HMI tags "Planchadora1"
   "Planchadora1_EstadoSsDer" : Byte = PLC Planchadora1.EstadoSsDer, 1 s
   "Planchadora1_EstadoSsIzq" : Byte = PLC Planchadora1.EstadoSsIzq, 1 s
   "Planchadora1_EstadoSSMed" : Byte = PLC Planchadora1.EstadoSSMed, 1 s
   "Planchadora1_FactorCorrRend" : Real = PLC Planchadora1.FactorCorrRend, 1 s
   "Planchadora1_FechaHoraPLC" : DTL = PLC Planchadora1.FechaHoraPLC, 1 s
   "Planchadora1_Operadores{1}_Estado" : Bool = PLC Planchadora1.Operadores[1].Estado, 1 s
   "Planchadora1_Operadores{1}_Produccion" : DInt = PLC Planchadora1.Operadores[1].Produccion, 1 s
   "Planchadora1_Operadores{1}_Rendimiento" : DInt = PLC Planchadora1.Operadores[1].Rendimiento, 1 s
   "Planchadora1_Operadores{1}_RendPesado" : DInt = PLC Planchadora1.Operadores[1].RendPesado, 1 s
   "Planchadora1_Operadores{1}_Tiempo" : DInt = PLC Planchadora1.Operadores[1].Tiempo, 1 s
   "Planchadora1_Operadores{10}_Estado" : Bool = PLC Planchadora1.Operadores[10].Estado, 1 s
   "Planchadora1_Operadores{10}_Produccion" : DInt = PLC Planchadora1.Operadores[10].Produccion, 1 s
   "Planchadora1_Operadores{10}_Rendimiento" : DInt = PLC Planchadora1.Operadores[10].Rendimiento, 1 s
   "Planchadora1_Operadores{10}_RendPesado" : DInt = PLC Planchadora1.Operadores[10].RendPesado AT %DB1.DBD0, 1 s
   "Planchadora1_Operadores{10}_Tiempo" : DInt = PLC Planchadora1.Operadores[10].Tiempo, 1 s
   "Planchadora1_Operadores{2}_Estado" : Bool = PLC Planchadora1.Operadores[2].Estado, 1 s
   "Planchadora1_Operadores{2}_Produccion" : DInt = PLC Planchadora1.Operadores[2].Produccion, 1 s
   "Planchadora1_Operadores{2}_Rendimiento" : DInt = PLC Planchadora1.Operadores[2].Rendimiento, 1 s
   "Planchadora1_Operadores{2}_RendPesado" : DInt = PLC Planchadora1.Operadores[2].RendPesado AT %DB1.DBD0, 1 s
   "Planchadora1_Operadores{2}_Tiempo" : DInt = PLC Planchadora1.Operadores[2].Tiempo, 1 s
   "Planchadora1_Operadores{3}_Estado" : Bool = PLC Planchadora1.Operadores[3].Estado, 1 s
   "Planchadora1_Operadores{3}_Produccion" : DInt = PLC Planchadora1.Operadores[3].Produccion, 1 s
   "Planchadora1_Operadores{3}_Rendimiento" : DInt = PLC Planchadora1.Operadores[3].Rendimiento, 1 s
   "Planchadora1_Operadores{3}_RendPesado" : DInt = PLC Planchadora1.Operadores[3].RendPesado AT %DB1.DBD0, 1 s
   "Planchadora1_Operadores{3}_Tiempo" : DInt = PLC Planchadora1.Operadores[3].Tiempo, 1 s
   "Planchadora1_Operadores{4}_Estado" : Bool = PLC Planchadora1.Operadores[4].Estado, 1 s
   "Planchadora1_Operadores{4}_Produccion" : DInt = PLC Planchadora1.Operadores[4].Produccion, 1 s
   "Planchadora1_Operadores{4}_Rendimiento" : DInt = PLC Planchadora1.Operadores[4].Rendimiento, 1 s
   "Planchadora1_Operadores{4}_RendPesado" : DInt = PLC Planchadora1.Operadores[4].RendPesado AT %DB1.DBD0, 1 s
   "Planchadora1_Operadores{4}_Tiempo" : DInt = PLC Planchadora1.Operadores[4].Tiempo, 1 s
   "Planchadora1_Operadores{5}_Estado" : Bool = PLC Planchadora1.Operadores[4].Estado, 1 s
   "Planchadora1_Operadores{5}_Produccion" : DInt = PLC Planchadora1.Operadores[4].Produccion, 1 s
   "Planchadora1_Operadores{5}_Rendimiento" : DInt = PLC Planchadora1.Operadores[4].Rendimiento, 1 s
   "Planchadora1_Operadores{5}_RendPesado" : DInt = PLC Planchadora1.Operadores[4].RendPesado AT %DB1.DBD0, 1 s
   "Planchadora1_Operadores{5}_Tiempo" : DInt = PLC Planchadora1.Operadores[4].Tiempo, 1 s
   "Planchadora1_Operadores{6}_Estado" : Bool = PLC Planchadora1.Operadores[6].Estado, 1 s
   "Planchadora1_Operadores{6}_Produccion" : DInt = PLC Planchadora1.Operadores[6].Produccion, 1 s
   "Planchadora1_Operadores{6}_Rendimiento" : DInt = PLC Planchadora1.Operadores[6].Rendimiento, 1 s
   "Planchadora1_Operadores{6}_RendPesado" : DInt = PLC Planchadora1.Operadores[6].RendPesado AT %DB1.DBD0, 1 s
   "Planchadora1_Operadores{6}_Tiempo" : DInt = PLC Planchadora1.Operadores[6].Tiempo, 1 s
   "Planchadora1_Operadores{7}_Estado" : Bool = PLC Planchadora1.Operadores[6].Estado, 1 s
   "Planchadora1_Operadores{7}_Produccion" : DInt = PLC Planchadora1.Operadores[6].Produccion, 1 s
   "Planchadora1_Operadores{7}_Rendimiento" : DInt = PLC Planchadora1.Operadores[7].Rendimiento, 1 s
   "Planchadora1_Operadores{7}_RendPesado" : DInt = PLC Planchadora1.Operadores[6].RendPesado AT %DB1.DBD0, 1 s
   "Planchadora1_WeekDay" : USInt = PLC Planchadora1.FechaHoraPLC.WEEKDAY AT %DB1.DBX0.0, 1 s
   "Planchadora1_TiempoTotal" : DInt = PLC Planchadora1.TiempoTotal, 1 s
   "Planchadora1_Supervisores{4}_Tiempo" : DInt = PLC Planchadora1.Supervisores[4].Tiempo, 1 s
   "Planchadora1_Supervisores{4}_RendPesado" : DInt = PLC Planchadora1.Supervisores[4].RendPesado AT %DB1.DBD0, 1 s
   "Planchadora1_Supervisores{4}_Rendimiento" : DInt = PLC Planchadora1.Supervisores[4].Rendimiento, 1 s
   "Planchadora1_Supervisores{4}_Produccion" : DInt = PLC Planchadora1.Supervisores[4].Produccion, 1 s
   "Planchadora1_Supervisores{4}_Estado" : Bool = PLC Planchadora1.Supervisores[4].Estado, 1 s
   "Planchadora1_Supervisores{4}_Diadelasemana{7}_Salida" : Time_Of_Day = PLC Planchadora1.Supervisores[4].Diadelasemana[7].Salida, 1 h
   "Planchadora1_Supervisores{4}_Diadelasemana{7}_Entrada" : Time_Of_Day = PLC Planchadora1.Supervisores[4].Diadelasemana[7].Entrada, 1 h
   "Planchadora1_Supervisores{4}_Diadelasemana{7}_CantOp" : Int = PLC Planchadora1.Supervisores[4].Diadelasemana[7].CantOp, 1 s
   "Planchadora1_Supervisores{4}_Diadelasemana{6}_Salida" : Time_Of_Day = PLC Planchadora1.Supervisores[4].Diadelasemana[6].Salida, 1 h
   "Planchadora1_Supervisores{4}_Diadelasemana{6}_Entrada" : Time_Of_Day = PLC Planchadora1.Supervisores[4].Diadelasemana[6].Entrada, 1 h
   "Planchadora1_Supervisores{4}_Diadelasemana{3}_CantOp" : Int = PLC Planchadora1.Supervisores[4].Diadelasemana[3].CantOp, 1 s
   "Planchadora1_Supervisores{4}_Diadelasemana{3}_Entrada" : Time_Of_Day = PLC Planchadora1.Supervisores[4].Diadelasemana[3].Entrada, 1 h
   "Planchadora1_Supervisores{4}_Diadelasemana{3}_Salida" : Time_Of_Day = PLC Planchadora1.Supervisores[4].Diadelasemana[3].Salida, 1 h
   "Planchadora1_Supervisores{4}_Diadelasemana{4}_CantOp" : Int = PLC Planchadora1.Supervisores[4].Diadelasemana[4].CantOp, 1 s
   "Planchadora1_Supervisores{4}_Diadelasemana{4}_Entrada" : Time_Of_Day = PLC Planchadora1.Supervisores[4].Diadelasemana[4].Entrada, 1 h
   "Planchadora1_Supervisores{4}_Diadelasemana{4}_Salida" : Time_Of_Day = PLC Planchadora1.Supervisores[4].Diadelasemana[4].Salida, 1 h
   "Planchadora1_Supervisores{4}_Diadelasemana{5}_CantOp" : Int = PLC Planchadora1.Supervisores[4].Diadelasemana[5].CantOp, 1 s
   "Planchadora1_Supervisores{4}_Diadelasemana{5}_Entrada" : Time_Of_Day = PLC Planchadora1.Supervisores[4].Diadelasemana[5].Entrada, 1 h
   "Planchadora1_Supervisores{4}_Diadelasemana{5}_Salida" : Time_Of_Day = PLC Planchadora1.Supervisores[4].Diadelasemana[5].Salida, 1 h
   "Planchadora1_Supervisores{4}_Diadelasemana{6}_CantOp" : Int = PLC Planchadora1.Supervisores[4].Diadelasemana[6].CantOp, 1 s
   "Planchadora1_Supervisores{3}_Diadelasemana{6}_Salida" : Time_Of_Day = PLC Planchadora1.Supervisores[3].Diadelasemana[6].Salida, 1 h
   "Planchadora1_Supervisores{3}_Diadelasemana{7}_CantOp" : Int = PLC Planchadora1.Supervisores[3].Diadelasemana[7].CantOp, 1 s
   "Planchadora1_Supervisores{3}_Diadelasemana{7}_Entrda" : Time_Of_Day = PLC Planchadora1.Supervisores[3].Diadelasemana[7].Entrada, 1 h
   "Planchadora1_Supervisores{3}_Diadelasemana{7}_Salida" : Time_Of_Day = PLC Planchadora1.Supervisores[3].Diadelasemana[7].Salida, 1 h
   "Planchadora1_Supervisores{3}_Estado" : Bool = PLC Planchadora1.Supervisores[3].Estado, 1 s
   "Planchadora1_Supervisores{3}_Produccion" : DInt = PLC Planchadora1.Supervisores[3].Produccion, 1 s
   "Planchadora1_Supervisores{3}_Rendimiento" : DInt = PLC Planchadora1.Supervisores[3].Rendimiento, 1 s
   "Planchadora1_Supervisores{3}_RendPesado" : DInt = PLC Planchadora1.Supervisores[3].RendPesado AT %DB1.DBD0, 1 s
   "Planchadora1_Supervisores{3}_Tiempo" : DInt = PLC Planchadora1.Supervisores[3].Tiempo, 1 s
   "Planchadora1_Supervisores{4}_Diadelasemana{1}_CantOp" : Int = PLC Planchadora1.Supervisores[4].Diadelasemana[1].CantOp, 1 s
   "Planchadora1_Supervisores{4}_Diadelasemana{1}_Entrada" : Time_Of_Day = PLC Planchadora1.Supervisores[4].Diadelasemana[1].Entrada, 1 h
   "Planchadora1_Supervisores{4}_Diadelasemana{1}_Salida" : Time_Of_Day = PLC Planchadora1.Supervisores[4].Diadelasemana[1].Salida, 1 h
   "Planchadora1_Supervisores{4}_Diadelasemana{2}_CantOp" : Int = PLC Planchadora1.Supervisores[4].Diadelasemana[2].CantOp, 1 s
   "Planchadora1_Supervisores{4}_Diadelasemana{2}_Entrada" : Time_Of_Day = PLC Planchadora1.Supervisores[4].Diadelasemana[2].Entrada, 1 h
   "Planchadora1_Supervisores{4}_Diadelasemana{2}_Salida" : Time_Of_Day = PLC Planchadora1.Supervisores[4].Diadelasemana[2].Salida, 1 h
   "Planchadora1_Supervisores{3}_Diadelasemana{1}_Salida" : Time_Of_Day = PLC Planchadora1.Supervisores[3].Diadelasemana[1].Salida, 1 h
   "Planchadora1_Supervisores{3}_Diadelasemana{2}_CantOp" : Int = PLC Planchadora1.Supervisores[3].Diadelasemana[2].CantOp, 1 s
   "Planchadora1_Supervisores{3}_Diadelasemana{2}_Entrda" : Time_Of_Day = PLC Planchadora1.Supervisores[3].Diadelasemana[2].Entrada, 1 h
   "Planchadora1_Supervisores{3}_Diadelasemana{2}_Salida" : Time_Of_Day = PLC Planchadora1.Supervisores[3].Diadelasemana[2].Salida, 1 h
   "Planchadora1_Supervisores{3}_Diadelasemana{3}_CantOp" : Int = PLC Planchadora1.Supervisores[3].Diadelasemana[3].CantOp, 1 s
   "Planchadora1_Supervisores{3}_Diadelasemana{3}_Entrda" : Time_Of_Day = PLC Planchadora1.Supervisores[3].Diadelasemana[3].Entrada, 1 h
   "Planchadora1_Supervisores{3}_Diadelasemana{3}_Salida" : Time_Of_Day = PLC Planchadora1.Supervisores[3].Diadelasemana[3].Salida, 1 h
   "Planchadora1_Supervisores{3}_Diadelasemana{4}_CantOp" : Int = PLC Planchadora1.Supervisores[3].Diadelasemana[4].CantOp, 1 s
   "Planchadora1_Supervisores{3}_Diadelasemana{4}_Entrda" : Time_Of_Day = PLC Planchadora1.Supervisores[3].Diadelasemana[4].Entrada, 1 h
   "Planchadora1_Supervisores{3}_Diadelasemana{4}_Salida" : Time_Of_Day = PLC Planchadora1.Supervisores[3].Diadelasemana[4].Salida, 1 h
   "Planchadora1_Supervisores{3}_Diadelasemana{5}_CantOp" : Int = PLC Planchadora1.Supervisores[3].Diadelasemana[5].CantOp, 1 s
   "Planchadora1_Supervisores{3}_Diadelasemana{5}_Entrda" : Time_Of_Day = PLC Planchadora1.Supervisores[3].Diadelasemana[5].Entrada, 1 h
   "Planchadora1_Supervisores{3}_Diadelasemana{5}_Salida" : Time_Of_Day = PLC Planchadora1.Supervisores[3].Diadelasemana[5].Salida, 1 h
   "Planchadora1_Supervisores{3}_Diadelasemana{6}_CantOp" : Int = PLC Planchadora1.Supervisores[3].Diadelasemana[6].CantOp, 1 s
   "Planchadora1_Supervisores{3}_Diadelasemana{6}_Entrda" : Time_Of_Day = PLC Planchadora1.Supervisores[3].Diadelasemana[6].Entrada, 1 h
   "Planchadora1_Supervisores{2}_Diadelasemana{6}_Entrda" : Time_Of_Day = PLC Planchadora1.Supervisores[2].Diadelasemana[6].Entrada, 1 h
   "Planchadora1_Supervisores{2}_Diadelasemana{6}_Salida" : Time_Of_Day = PLC Planchadora1.Supervisores[2].Diadelasemana[6].Salida, 1 h
   "Planchadora1_Supervisores{2}_Diadelasemana{7}_CantOp" : Int = PLC Planchadora1.Supervisores[2].Diadelasemana[7].CantOp, 1 s
   "Planchadora1_Supervisores{2}_Diadelasemana{7}_Entrda" : Time_Of_Day = PLC Planchadora1.Supervisores[2].Diadelasemana[7].Entrada, 1 h
   "Planchadora1_Supervisores{2}_Diadelasemana{7}_Salida" : Time_Of_Day = PLC Planchadora1.Supervisores[2].Diadelasemana[7].Salida, 1 h
   "Planchadora1_Supervisores{2}_Estado" : Bool = PLC Planchadora1.Supervisores[2].Estado, 1 s
   "Planchadora1_Supervisores{2}_Produccion" : DInt = PLC Planchadora1.Supervisores[2].Produccion, 1 s
   "Planchadora1_Supervisores{2}_Rendimiento" : DInt = PLC Planchadora1.Supervisores[2].Rendimiento, 1 s
   "Planchadora1_Supervisores{2}_RendPesado" : DInt = PLC Planchadora1.Supervisores[2].RendPesado AT %DB1.DBD0, 1 s
   "Planchadora1_Supervisores{2}_Tiempo" : DInt = PLC Planchadora1.Supervisores[2].Tiempo, 1 s
   "Planchadora1_Supervisores{3}_Diadelasemana{1}_CantOp" : Int = PLC Planchadora1.Supervisores[3].Diadelasemana[1].CantOp, 1 s
   "Planchadora1_Supervisores{3}_Diadelasemana{1}_Entrda" : Time_Of_Day = PLC Planchadora1.Supervisores[3].Diadelasemana[1].Entrada, 1 h
   "Planchadora1_Supervisores{2}_Diadelasemana{2}_Entrda" : Time_Of_Day = PLC Planchadora1.Supervisores[2].Diadelasemana[2].Entrada, 1 h
   "Planchadora1_Supervisores{2}_Diadelasemana{2}_Salida" : Time_Of_Day = PLC Planchadora1.Supervisores[2].Diadelasemana[2].Salida, 1 h
   "Planchadora1_Supervisores{2}_Diadelasemana{3}_CantOp" : Int = PLC Planchadora1.Supervisores[2].Diadelasemana[3].CantOp, 1 s
   "Planchadora1_Supervisores{2}_Diadelasemana{3}_Entrda" : Time_Of_Day = PLC Planchadora1.Supervisores[2].Diadelasemana[3].Entrada, 1 h
   "Planchadora1_Supervisores{2}_Diadelasemana{3}_Salida" : Time_Of_Day = PLC Planchadora1.Supervisores[2].Diadelasemana[3].Salida, 1 h
   "Planchadora1_Supervisores{2}_Diadelasemana{4}_CantOp" : Int = PLC Planchadora1.Supervisores[2].Diadelasemana[4].CantOp, 1 s
   "Planchadora1_Supervisores{2}_Diadelasemana{4}_Entrda" : Time_Of_Day = PLC Planchadora1.Supervisores[2].Diadelasemana[4].Entrada, 1 h
   "Planchadora1_Supervisores{2}_Diadelasemana{4}_Salida" : Time_Of_Day = PLC Planchadora1.Supervisores[2].Diadelasemana[4].Salida, 1 h
   "Planchadora1_Supervisores{2}_Diadelasemana{5}_CantOp" : Int = PLC Planchadora1.Supervisores[2].Diadelasemana[5].CantOp, 1 s
   "Planchadora1_Supervisores{2}_Diadelasemana{5}_Entrda" : Time_Of_Day = PLC Planchadora1.Supervisores[2].Diadelasemana[5].Entrada, 1 h
   "Planchadora1_Supervisores{2}_Diadelasemana{5}_Salida" : Time_Of_Day = PLC Planchadora1.Supervisores[2].Diadelasemana[5].Salida, 1 h
   "Planchadora1_Supervisores{2}_Diadelasemana{6}_CantOp" : Int = PLC Planchadora1.Supervisores[2].Diadelasemana[6].CantOp, 1 s
   "Planchadora1_Supervisores{1}_Diadelasemana{6}_CantOp" : Int = PLC Planchadora1.Supervisores[1].Diadelasemana[6].CantOp, 1 s
   "Planchadora1_Supervisores{1}_Diadelasemana{6}_Entrda" : Time_Of_Day = PLC Planchadora1.Supervisores[1].Diadelasemana[6].Entrada, 1 h
   "Planchadora1_Supervisores{1}_Diadelasemana{6}_Salida" : Time_Of_Day = PLC Planchadora1.Supervisores[1].Diadelasemana[6].Salida, 1 h
   "Planchadora1_Supervisores{1}_Diadelasemana{7}_CantOp" : Int = PLC Planchadora1.Supervisores[1].Diadelasemana[7].CantOp, 1 s
   "Planchadora1_Supervisores{1}_Diadelasemana{7}_Entrda" : Time_Of_Day = PLC Planchadora1.Supervisores[1].Diadelasemana[7].Entrada, 1 h
   "Planchadora1_Supervisores{1}_Diadelasemana{7}_Salida" : Time_Of_Day = PLC Planchadora1.Supervisores[1].Diadelasemana[7].Salida, 1 h
   "Planchadora1_Supervisores{1}_Estado" : Bool = PLC Planchadora1.Supervisores[1].Estado, 1 s
   "Planchadora1_Supervisores{1}_Produccion" : DInt = PLC Planchadora1.Supervisores[1].Produccion, 1 s
   "Planchadora1_Supervisores{1}_Rendimiento" : DInt = PLC Planchadora1.Supervisores[1].Rendimiento, 1 s
   "Planchadora1_Supervisores{1}_RendPesado" : DInt = PLC Planchadora1.Supervisores[1].RendPesado AT %DB1.DBD0, 1 s
   "Planchadora1_Supervisores{1}_Tiempo" : DInt = PLC Planchadora1.Supervisores[1].Tiempo, 1 s
   "Planchadora1_Supervisores{2}_Diadelasemana{1}_CantOp" : Int = PLC Planchadora1.Supervisores[2].Diadelasemana[1].CantOp, 1 s
   "Planchadora1_Supervisores{2}_Diadelasemana{1}_Entrda" : Time_Of_Day = PLC Planchadora1.Supervisores[2].Diadelasemana[1].Entrada, 1 h
   "Planchadora1_Supervisores{2}_Diadelasemana{1}_Salida" : Time_Of_Day = PLC Planchadora1.Supervisores[2].Diadelasemana[1].Salida, 1 h
   "Planchadora1_Supervisores{2}_Diadelasemana{2}_CantOp" : Int = PLC Planchadora1.Supervisores[2].Diadelasemana[2].CantOp, 1 s
   "Planchadora1_Supervisores{1}_Diadelasemana{1}_CantOp" : Int = PLC Planchadora1.Supervisores[1].Diadelasemana[1].CantOp, 1 s
   "Planchadora1_Supervisores{1}_Diadelasemana{1}_Entrda" : Time_Of_Day = PLC Planchadora1.Supervisores[1].Diadelasemana[1].Entrada, 1 h
   "Planchadora1_Supervisores{1}_Diadelasemana{1}_Salida" : Time_Of_Day = PLC Planchadora1.Supervisores[1].Diadelasemana[1].Salida, 1 h
   "Planchadora1_Supervisores{1}_Diadelasemana{2}_CantOp" : Int = PLC Planchadora1.Supervisores[1].Diadelasemana[2].CantOp, 1 s
   "Planchadora1_Supervisores{1}_Diadelasemana{2}_Entrda" : Time_Of_Day = PLC Planchadora1.Supervisores[1].Diadelasemana[2].Entrada, 1 h
   "Planchadora1_Supervisores{1}_Diadelasemana{2}_Salida" : Time_Of_Day = PLC Planchadora1.Supervisores[1].Diadelasemana[2].Salida, 1 h
   "Planchadora1_Supervisores{1}_Diadelasemana{3}_CantOp" : Int = PLC Planchadora1.Supervisores[1].Diadelasemana[3].CantOp, 1 s
   "Planchadora1_Supervisores{1}_Diadelasemana{3}_Entrda" : Time_Of_Day = PLC Planchadora1.Supervisores[1].Diadelasemana[3].Entrada, 1 h
   "Planchadora1_Supervisores{1}_Diadelasemana{3}_Salida" : Time_Of_Day = PLC Planchadora1.Supervisores[1].Diadelasemana[3].Salida, 1 h
   "Planchadora1_Supervisores{1}_Diadelasemana{4}_CantOp" : Int = PLC Planchadora1.Supervisores[1].Diadelasemana[4].CantOp, 1 s
   "Planchadora1_Supervisores{1}_Diadelasemana{4}_Entrda" : Time_Of_Day = PLC Planchadora1.Supervisores[1].Diadelasemana[4].Entrada, 1 h
   "Planchadora1_Supervisores{1}_Diadelasemana{4}_Salida" : Time_Of_Day = PLC Planchadora1.Supervisores[1].Diadelasemana[4].Salida, 1 h
   "Planchadora1_Supervisores{1}_Diadelasemana{5}_CantOp" : Int = PLC Planchadora1.Supervisores[1].Diadelasemana[5].CantOp, 1 s
   "Planchadora1_Supervisores{1}_Diadelasemana{5}_Entrda" : Time_Of_Day = PLC Planchadora1.Supervisores[1].Diadelasemana[5].Entrada, 1 h
   "Planchadora1_Supervisores{1}_Diadelasemana{5}_Salida" : Time_Of_Day = PLC Planchadora1.Supervisores[1].Diadelasemana[5].Salida, 1 h
   "Planchadora1_Rendimiento_100" : Real = PLC Planchadora1.Rendimiento_100, 1 s
   "Planchadora1_Rendimiento_Amarillo" : Real = PLC Planchadora1.Productividad_Amarillo, 1 s
   "Planchadora1_Rendimiento_Rojo" : Real = PLC Planchadora1.Rendimiento_Rojo, 1 s
   "Planchadora1_Rendimiento_Verde" : Real = PLC Planchadora1.Productividad_Verde, 1 s
   "Planchadora1_RendimientoCada15" : DInt = PLC Planchadora1.RendimientoCada15, 1 s
   "Planchadora1_RendimientoTotal" : DInt = PLC Planchadora1.RendimientoTotal, 1 s
   "Planchadora1_RendPesado" : DInt = PLC Planchadora1.RendPesado AT %DB1.DBD0, 1 s
   "Planchadora1_RendPesado_100" : Real = PLC Planchadora1.RendPesado_100, 1 s
   "Planchadora1_SumaOperario" : Int = PLC Planchadora1.SumaOperario AT %DB1.DBX0.0, 10 s
      on ChangeValue: "S407_Act_IndicePLC"()
   "Planchadora1_Operadores{8}_Estado" : Bool = PLC Planchadora1.Operadores[8].Estado, 1 s
   "Planchadora1_Operadores{8}_Produccion" : DInt = PLC Planchadora1.Operadores[8].Produccion, 1 s
   "Planchadora1_Operadores{8}_Rendimiento" : DInt = PLC Planchadora1.Operadores[8].Rendimiento, 1 s
   "Planchadora1_Operadores{8}_RendPesado" : DInt = PLC Planchadora1.Operadores[8].RendPesado AT %DB1.DBD0, 1 s
   "Planchadora1_Operadores{8}_Tiempo" : DInt = PLC Planchadora1.Operadores[8].Tiempo, 1 s
   "Planchadora1_Operadores{9}_Estado" : Bool = PLC Planchadora1.Operadores[9].Estado, 1 s
   "Planchadora1_Operadores{9}_Produccion" : DInt = PLC Planchadora1.Operadores[9].Produccion, 1 s
   "Planchadora1_Operadores{9}_Rendimiento" : DInt = PLC Planchadora1.Operadores[9].Rendimiento, 1 s
   "Planchadora1_Operadores{9}_RendPesado" : DInt = PLC Planchadora1.Operadores[9].RendPesado AT %DB1.DBD0, 1 s
   "Planchadora1_Operadores{9}_Tiempo" : DInt = PLC Planchadora1.Operadores[9].Tiempo, 1 s
   "Planchadora1_Productividad" : DInt = PLC Planchadora1.Productividad, 1 s
   "Planchadora1_Productividad_100" : Real = PLC Planchadora1.Productividad_100, 1 s
   "Planchadora1_Productividad_Amarillo" : Real = PLC Planchadora1.Productividad_Amarillo, 1 s
   "Planchadora1_Productividad_Rojo" : Real = PLC Planchadora1.Productividad_Rojo, 1 s
   "Planchadora1_Productividad_Verde" : Real = PLC Planchadora1.Productividad_Verde, 1 s
   "Planchadora1_ProductividadCada15" : DInt = PLC Planchadora1.ProductividadCada15, 1 s
   "Planchadora1_ProductividadTotal" : DInt = PLC Planchadora1.ProductividadTotal, 1 s
   "Planchadora1_Rendimiento" : DInt = PLC Planchadora1.Rendimiento, 1 s
   "Planchadora1_Operadores{7}_Tiempo" : DInt = PLC Planchadora1.Operadores[7].Tiempo, 1 s

HMI tags "Planchadora2"
   "Planchadora2_WeekDay_Int" : Int AT %DB1.DBX0.0
   "Planchadora2_Supervisores{1}_Tiempo" : DInt = PLC Planchadora2.Supervisores[1].Tiempo, 1 s
   "Planchadora2_Supervisores{2}_Estado" : Bool = PLC Planchadora2.Supervisores[2].Estado, 1 s
   "Planchadora2_Supervisores{2}_Produccion" : DInt = PLC Planchadora2.Supervisores[2].Produccion, 1 s
   "Planchadora2_Supervisores{2}_Rendimiento" : DInt = PLC Planchadora2.Supervisores[2].Rendimiento, 1 s
   "Planchadora2_Supervisores{2}_RendPesado" : DInt = PLC Planchadora2.Supervisores[2].RendPesado AT %DB1.DBD0, 1 s
   "Planchadora2_Supervisores{2}_Tiempo" : DInt = PLC Planchadora2.Supervisores[2].Tiempo, 1 s
   "Planchadora2_Supervisores{3}_Estado" : Bool = PLC Planchadora2.Supervisores[3].Estado, 1 s
   "Planchadora2_Supervisores{3}_Produccion" : DInt = PLC Planchadora2.Supervisores[3].Produccion, 1 s
   "Planchadora2_Supervisores{3}_Rendimiento" : DInt = PLC Planchadora2.Supervisores[3].Rendimiento, 1 s
   "Planchadora2_Supervisores{3}_RendPesado" : DInt = PLC Planchadora2.Supervisores[3].RendPesado AT %DB1.DBD0, 1 s
   "Planchadora2_Supervisores{3}_Tiempo" : DInt = PLC Planchadora2.Supervisores[3].Tiempo, 1 s
   "Planchadora2_Supervisores{4}_Estado" : Bool = PLC Planchadora2.Supervisores[4].Estado, 1 s
   "Planchadora2_Supervisores{4}_Produccion" : DInt = PLC Planchadora2.Supervisores[4].Produccion, 1 s
   "Planchadora2_Supervisores{4}_Rendimiento" : DInt = PLC Planchadora2.Supervisores[4].Rendimiento, 1 s
   "Planchadora2_Supervisores{4}_RendPesado" : DInt = PLC Planchadora2.Supervisores[4].RendPesado AT %DB1.DBD0, 1 s
   "Planchadora2_Supervisores{4}_Tiempo" : DInt = PLC Planchadora2.Supervisores[4].Tiempo, 1 s
   "Planchadora2_TiempoTotal" : DInt = PLC Planchadora2.TiempoTotal, 1 s
   "Planchadora2_WeekDay" : USInt = PLC Planchadora2.FechaHoraPLC.WEEKDAY AT %DB1.DBB0, 1 s
   "Planchadora2_Operadores{9}_RendPesado" : DInt = PLC Planchadora2.Operadores[9].RendPesado AT %DB1.DBD0, 1 s
   "Planchadora2_Operadores{9}_Tiempo" : DInt = PLC Planchadora2.Operadores[9].Tiempo, 1 s
   "Planchadora2_Productividad_100" : Real = PLC Planchadora2.Productividad_100, 1 s
   "Planchadora2_ProductividadCada15" : DInt = PLC Planchadora2.ProductividadCada15, 1 s
   "Planchadora2_ProductividadTotal" : DInt = PLC Planchadora2.ProductividadTotal, 1 s
   "Planchadora2_Rendimiento_100" : Real = PLC Planchadora2.Rendimiento_100, 1 s
   "Planchadora2_RendimientoCada15" : DInt = PLC Planchadora2.RendimientoCada15, 1 s
   "Planchadora2_RendimientoTotal" : DInt = PLC Planchadora2.RendimientoTotal, 1 s
   "Planchadora2_RendPesado" : DInt = PLC Planchadora2.RendPesado AT %DB1.DBD0, 1 s
   "Planchadora2_RendPesado_100" : Real = PLC Planchadora2.RendPesado_100, 1 s
   "Planchadora2_SumaOperario" : Int = PLC Planchadora2.SumaOperario AT %DB1.DBX0.0, 1 s
   "Planchadora2_Supervisores{1}_Estado" : Bool = PLC Planchadora2.Supervisores[1].Estado, 1 s
   "Planchadora2_Supervisores{1}_Produccion" : DInt = PLC Planchadora2.Supervisores[1].Produccion, 1 s
   "Planchadora2_Supervisores{1}_Rendimiento" : DInt = PLC Planchadora2.Supervisores[1].Rendimiento, 1 s
   "Planchadora2_Supervisores{1}_RendPesado" : DInt = PLC Planchadora2.Supervisores[1].RendPesado AT %DB1.DBD0, 1 s
   "Planchadora2_Operadores{6}_Produccion" : DInt = PLC Planchadora2.Operadores[6].Produccion, 1 s
   "Planchadora2_Operadores{6}_Rendimiento" : DInt = PLC Planchadora2.Operadores[6].Rendimiento, 1 s
   "Planchadora2_Operadores{6}_RendPesado" : DInt = PLC Planchadora2.Operadores[6].RendPesado AT %DB1.DBD0, 1 s
   "Planchadora2_Operadores{6}_Tiempo" : DInt = PLC Planchadora2.Operadores[6].Tiempo, 1 s
   "Planchadora2_Operadores{7}_Estado" : Bool = PLC Planchadora2.Operadores[7].Estado, 1 s
   "Planchadora2_Operadores{7}_Produccion" : DInt = PLC Planchadora2.Operadores[7].Produccion, 1 s
   "Planchadora2_Operadores{7}_Rendimiento" : DInt = PLC Planchadora2.Operadores[7].Rendimiento, 1 s
   "Planchadora2_Operadores{7}_RendPesado" : DInt = PLC Planchadora2.Operadores[7].RendPesado AT %DB1.DBD0, 1 s
   "Planchadora2_Operadores{7}_Tiempo" : DInt = PLC Planchadora2.Operadores[7].Tiempo, 1 s
   "Planchadora2_Operadores{8}_Estado" : Bool = PLC Planchadora2.Operadores[8].Estado, 1 s
   "Planchadora2_Operadores{8}_Produccion" : DInt = PLC Planchadora2.Operadores[8].Produccion, 1 s
   "Planchadora2_Operadores{8}_Rendimiento" : DInt = PLC Planchadora2.Operadores[8].Rendimiento, 1 s
   "Planchadora2_Operadores{8}_RendPesado" : DInt = PLC Planchadora2.Operadores[8].RendPesado, 1 s
   "Planchadora2_Operadores{8}_Tiempo" : DInt = PLC Planchadora2.Operadores[8].Tiempo, 1 s
   "Planchadora2_Operadores{9}_Estado" : Bool = PLC Planchadora2.Operadores[9].Estado, 1 s
   "Planchadora2_Operadores{9}_Produccion" : DInt = PLC Planchadora2.Operadores[9].Produccion, 1 s
   "Planchadora2_Operadores{9}_Rendimiento" : DInt = PLC Planchadora2.Operadores[9].Rendimiento, 1 s
   "Planchadora2_Operadores{2}_RendPesado" : DInt = PLC Planchadora2.Operadores[2].RendPesado AT %DB1.DBD0, 1 s
   "Planchadora2_Operadores{2}_Tiempo" : DInt = PLC Planchadora2.Operadores[3].Tiempo, 1 s
   "Planchadora2_Operadores{3}_Estado" : Bool = PLC Planchadora2.Operadores[3].Estado, 1 s
   "Planchadora2_Operadores{3}_Produccion" : DInt = PLC Planchadora2.Operadores[3].Produccion, 1 s
   "Planchadora2_Operadores{3}_Rendimiento" : DInt = PLC Planchadora2.Operadores[3].Rendimiento, 1 s
   "Planchadora2_Operadores{3}_RendPesado" : DInt = PLC Planchadora2.Operadores[3].RendPesado AT %DB1.DBD0, 1 s
   "Planchadora2_Operadores{3}_Tiempo" : DInt = PLC Planchadora2.Operadores[3].Tiempo, 1 s
   "Planchadora2_Operadores{4}_Estado" : Bool = PLC Planchadora2.Operadores[4].Estado, 1 s
   "Planchadora2_Operadores{4}_Produccion" : DInt = PLC Planchadora2.Operadores[4].Produccion, 1 s
   "Planchadora2_Operadores{4}_Rendimiento" : DInt = PLC Planchadora2.Operadores[5].Rendimiento, 1 s
   "Planchadora2_Operadores{4}_RendPesado" : DInt = PLC Planchadora2.Operadores[5].RendPesado AT %DB1.DBD0, 1 s
   "Planchadora2_Operadores{4}_Tiempo" : DInt = PLC Planchadora2.Operadores[5].Tiempo, 1 s
   "Planchadora2_Operadores{5}_Estado" : Bool = PLC Planchadora2.Operadores[5].Estado, 1 s
   "Planchadora2_Operadores{5}_Produccion" : DInt = PLC Planchadora2.Operadores[5].Produccion, 1 s
   "Planchadora2_Operadores{5}_Rendimiento" : DInt = PLC Planchadora2.Operadores[5].Rendimiento, 1 s
   "Planchadora2_Operadores{5}_RendPesado" : DInt = PLC Planchadora2.Operadores[5].RendPesado AT %DB1.DBD0, 1 s
   "Planchadora2_Operadores{5}_Tiempo" : DInt = PLC Planchadora2.Operadores[5].Tiempo, 1 s
   "Planchadora2_Operadores{6}_Estado" : Bool = PLC Planchadora2.Operadores[6].Estado, 1 s
   "Planchadora2_EstadoSsIzq" : Byte = PLC Planchadora2.EstadoSsIzq, 1 s
   "Planchadora2_EstadoSSMed" : Byte = PLC Planchadora2.EstadoSSMed, 1 s
   "Planchadora2_Operadores{1}_Estado" : Bool = PLC Planchadora2.Operadores[1].Estado, 1 s
   "Planchadora2_Operadores{1}_Produccion" : DInt = PLC Planchadora2.Operadores[1].Produccion, 1 s
   "Planchadora2_Operadores{1}_Productividad" : DInt = PLC Planchadora2.Operadores[1].Productividad, 1 s
   "Planchadora2_Operadores{1}_Rendimiento" : DInt = PLC Planchadora2.Operadores[1].Rendimiento, 1 s
   "Planchadora2_Operadores{1}_RendPesado" : DInt = PLC Planchadora2.Operadores[1].RendPesado AT %DB1.DBD0, 1 s
   "Planchadora2_Operadores{1}_Tiempo" : DInt = PLC Planchadora2.Operadores[1].Tiempo, 1 s
   "Planchadora2_Operadores{10}_Estado" : Bool = PLC Planchadora2.Operadores[10].Estado, 1 s
   "Planchadora2_Operadores{10}_Produccion" : DInt = PLC Planchadora2.Operadores[10].Produccion, 1 s
   "Planchadora2_Operadores{10}_Rendimiento" : DInt = PLC Planchadora2.Operadores[10].Rendimiento, 1 s
   "Planchadora2_Operadores{10}_RendPesado" : DInt = PLC Planchadora2.Operadores[10].RendPesado AT %DB1.DBD0, 1 s
   "Planchadora2_Operadores{10}_Tiempo" : DInt = PLC Planchadora2.Operadores[10].Tiempo, 1 s
   "Planchadora2_Operadores{2}_Estado" : Bool = PLC Planchadora2.Operadores[2].Estado, 1 s
   "Planchadora2_Operadores{2}_Produccion" : DInt = PLC Planchadora2.Operadores[2].Produccion, 1 s
   "Planchadora2_Operadores{2}_Rendimiento" : DInt = PLC Planchadora2.Operadores[2].Rendimiento, 1 s
   "Plan2EnProd" : Bool = PLC Plan2EnProd AT %M4.3, 1 s
   "Planchadora2_EstadoSsDer" : Byte = PLC Planchadora2.EstadoSsDer, 1 s

HMI tags "Lavadora1"
   "Lav1_Programa" : Int AT 4x403158, 2 s
   "Lav1_Operador" : Int AT 4x403155, 2 s
      on ChangeValue: "S304_ActualizarOpEnPrincipal"(1)
   "Lav1_Alarma" : Bit AT 0x2057, 2 s
   "Lav1_CantRopa" : Int AT 4x403157, 2 s
   "Lav1_GrabarBDD" : Bit AT 0x3244, 1 s
      on ChangeValue: "S14_Write_data_Lav1"()
   "Lav1_FchFin_Ano" : Int AT 4x403172, 500 ms
   "Lav1_FchFin_Mes" : Int AT 4x403171, 500 ms
   "Lav1_FchFin_Dia" : Int AT 4x403170, 500 ms
   "Lav1_FchFin_Hr" : Int AT 4x403169, 500 ms
   "Lav1_FchFin_Min" : Int AT 4x403168, 500 ms
   "Lav1_FchFin_Seg" : Int AT 4x403167, 500 ms
   "Lav1_FchIni_Ano" : Int AT 4x403166, 1 s
   "Lav1_FchIni_Mes" : Int AT 4x403165, 1 s
   "Lav1_FchIni_Dia" : Int AT 4x403164, 1 s
   "Lav1_FchIni_Hr" : Int AT 4x403163, 1 s
   "Lav1_FchIni_Min" : Int AT 4x403162, 1 s
   "Lav1_FchIni_Seg" : Int AT 4x403161, 1 s
   "Lav1_Cliente_0" : Int AT 4x403160, 2 s
      on ChangeValue: "S104_ActualizarCliEmPrincipal"(1, 0)
   "Lav1_CicloValido" : Bit AT 0x3208, 100 ms
   "Lav1_Operador_Str" : WString[64], internal
   "Lav1_Cliente_1" : Int AT 4x403174, 2 s
      on ChangeValue: "S104_ActualizarCliEmPrincipal"(1, 1)
   "Lav1_Cliente_2" : Int AT 4x403176, 2 s
      on ChangeValue: "S104_ActualizarCliEmPrincipal"(1, 2)
   "Lav1_Fch_segs" : Int AT 4x404087, 500 ms
   "Lav1_Fch_Mins" : Int AT 4x404088, 500 ms
   "Lav1_Fch_Hr" : Int AT 4x404089, 500 ms
   "Lav1_Fch_Dia" : Int AT 4x404091, 500 ms
   "Lav1_Fch_Mes" : Int AT 4x404092, 500 ms
   "Lav1_Fch_Ano" : Int AT 4x404093, 500 ms
   "Lav1_Cliente_0_PLC" : Int AT 4x403159, 2 s
   "Lav1_Cliente_1_PLC" : Int AT 4x403173, 2 s
   "Lav1_Cliente_2_PLC" : Int AT 4x403175, 2 s
   "Lav1_Operador_PLC" : Int AT 4x403154, 2 s
      on ChangeValue: "S304_ActualizarOpEnPrincipal"(1)
   "Lav1_CantR_PLC" : Int AT 4x403156, 2 s
   "Lav1_AlarmaVibracion" : Bit AT 0x3390, 2 s
      on ChangeValue: "SA1_email_Vibr"(); "S40_Write_Fall1BDD"()
   "Lav1_EnCiclo" : Bit AT 0x3081, 1 s
      on ChangeValue: "SA3_Act_HoraFinEstPrincLav1"()
   "Lav1_CicloFinalizado" : Bit AT 0x3251, 2 s
   "Lav1_Ciclograbado" : Bit AT 0x3231, 1 s
   "Lav1_ComienzoCiclo" : Bit AT 0x3230, 1 s
   "Lav1_Falla" : Int AT 4x403183, 500 ms
   "Lav1_ConfFalla" : Bit AT 0x3252, 1 s
   "Lav1_PulsParadaPres" : Bit AT 0x3253, 1 s
      on ChangeValue: "S40_Write_Fall1BDD"()
   "Lav1_Cli_0_Str" : WString[64], internal
   "Lav1_Cli_1_Str" : WString[64], internal
   "Lav1_Cli_2_Str" : WString[64], internal
   "Lav1_FinEstimado_Panel" : DateTime, internal
   "Lav1_ProgAGrabar" : Int AT 4x401025, 2 s
   "Lav1_PulsParadaPres_1" : Bit AT 0x3254, 1 s
   "Lav1_Cont_IntentosGrabado" : Int, internal
   "Lav1_X0_iPres_SinAire" : Bit AT 0x2049, 1 s
   "Lav1_X1_iPres_Freno" : Bit AT 0x2050, 1 s
   "Lav1_X2_iTermico" : Bit AT 0x2051, 1 s
   "Lav1_X3_iSns_PCarga" : Bit AT 0x2052, 1 s
   "Lav1_X4_iSns_PDesc" : Bit AT 0x2053, 1 s
   "Lav1_X5_iPuls_DestrPuerta" : Bit AT 0x2054, 1 s
   "Lav1_X6_iSwitch_Vibra" : Bit AT 0x2055, 1 s
   "Lav1_X7_iFallVar" : Bit AT 0x2056, 1 s
   "Lav1_X11_iPulsMarcha" : Bit AT 0x2058, 1 s
   "Lav1_X12_iPulsPausa" : Bit AT 0x2059, 1 s
   "Lav1_X13_iNivBajo" : Bit AT 0x2060, 1 s
   "Lav1_X14_iBuscPtaCargArr" : Bit AT 0x2061, 1 s
   "Lav1_X15_iBuscPtaCargAba" : Bit AT 0x2062, 1 s
   "Lav1_X16_iBuscPtaDescArr" : Bit AT 0x2063, 1 s
   "Lav1_X17_iBuscPtaDescAba" : Bit AT 0x2064, 1 s
   "Lav1_X20_BloqMarchDesc" : Bit AT 0x2065, 1 s
   "Lav1_X21_iNiv_Alto" : Bit AT 0x2066, 1 s
   "Lav1_X22_iSns_Ind" : Bit AT 0x2067, 1 s
   "Lav1_X23_iPE" : Bit AT 0x2068, 1 s
   "Lav1_Y100_MachineOn" : Bit AT 1x102113, 1 s
   "Lav1_Y101_DosifPreLav" : Bit AT 1x102114, 1 s
   "Lav1_Y102_AvEjFinalNro2" : Bit AT 1x102115, 1 s
   "Lav1_Y103_AvEjFinalNro3" : Bit AT 1x102116, 1 s
   "Lav1_Y104_AvDosifLavNro1" : Bit AT 1x102117, 1 s
   "Lav1_Y105_Cloro_AvDosifL2" : Bit AT 1x102118, 1 s
   "Lav1_St_EnjIni" : Bit AT 0x3122, 1 s
   "Lav1_St_PrimLAv" : Bit AT 0x3127, 1 s
   "Lav1_St_SegLav" : Bit AT 0x3138, 1 s
   "Lav1_St_EnjFin" : Bit AT 0x3131, 1 s
   "Lav1_St_EspCentr" : Bit AT 0x3133, 1 s
   "Lav1_St_Centr" : Bit AT 0x3134, 1 s
   "Lav1_St_FrenoMaquina" : Bit AT 0x3135, 1 s
   "Lav1_St_PreLav" : Bit AT 0x3125, 1 s
   "Lav1_Programa_Anterior" : Int, internal
   "Lav1_grabFalla" : Bit AT 0x3253, 1 s
      on ChangeValue: "S40_Write_Fall1BDD"()
   "Lav1_CicloValido_CN" : Bit AT 0x3209, 1 s
   "Lav1_St_Ciclo" : Int AT 4x403182, 1 s
   "Lav1_FchFll_Ano" : Int AT 4x403198, 1 s
   "Lav1_FchFll_Mes" : Int AT 4x403197, 1 s
   "Lav1_FchFll_Dia" : Int AT 4x403196, 1 s
   "Lav1_FchFll_Hr" : Int AT 4x403195, 1 s
   "Lav1_FchFll_Mins" : Int AT 4x403194, 1 s
   "Lav1_FchFll_segs" : Int AT 4x403193, 1 s

HMI tags "Lavadora2"
   "Lav2_CantRopa" : Int AT 4x403157, 2 s
   "Lav2_GrabarBDD" : Bit AT 0x3244, 2 s
      on ChangeValue: "S15_Write_data_Lav2"()
   "Lav2_Alarma" : Bit AT 0x2057, 2 s
   "Lav2_Programa" : Int AT 4x403158, 2 s
   "Lav2_Operador" : Int AT 4x403155, 2 s
      on ChangeValue: "S304_ActualizarOpEnPrincipal"(2)
   "Lav2_FchFin_Ano" : Int AT 4x403172, 500 ms
   "Lav2_FchFin_Mes" : Int AT 4x403171, 500 ms
   "Lav2_FchFin_Dia" : Int AT 4x403170, 500 ms
   "Lav2_FchFin_Hr" : Int AT 4x403169, 500 ms
   "Lav2_FchFin_Min" : Int AT 4x403168, 500 ms
   "Lav2_FchFin_Seg" : Int AT 4x403167, 500 ms
   "Lav2_FchIni_Ano" : Int AT 4x403166, 1 s
   "Lav2_FchIni_Mes" : Int AT 4x403165, 1 s
   "Lav2_FchIni_Dia" : Int AT 4x403164, 1 s
   "Lav2_FchIni_Hr" : Int AT 4x403163, 1 s
   "Lav2_FchIni_Min" : Int AT 4x403162, 1 s
   "Lav2_FchIni_Seg" : Int AT 4x403161, 1 s
   "Lav2_Cliente_0" : Int AT 4x403160, 2 s
      on ChangeValue: "S104_ActualizarCliEmPrincipal"(2, 0)
   "Lav2_CicloValido" : Bit AT 0x3208, 100 ms
   "Lav2_Operador_Str" : WString[64], internal
   "Lav2_Cliente_1" : Int AT 4x403174, 2 s
      on ChangeValue: "S104_ActualizarCliEmPrincipal"(2, 1)
   "Lav2_Cliente_2" : Int AT 4x403176, 2 s
      on ChangeValue: "S104_ActualizarCliEmPrincipal"(2, 2)
   "Lav2_Fch_Mins" : Int AT 4x404088, 500 ms
   "Lav2_Fch_Hr" : Int AT 4x404089, 500 ms
   "Lav2_Fch_segs" : Int AT 4x404087, 500 ms
   "Lav2_Fch_Dia" : Int AT 4x404091, 500 ms
   "Lav2_Fch_Mes" : Int AT 4x404092, 500 ms
   "Lav2_Fch_Ano" : Int AT 4x404093, 500 ms
   "Lav2_CantRopa_PLC" : Int AT 4x403156, 2 s
   "Lav2_Cliente_0_PLC" : Int AT 4x403159, 2 s
   "Lav2_Cliente_1_PLC" : Int AT 4x403173, 2 s
   "Lav2_Cliente_2_PLC" : Int AT 4x403175, 2 s
   "Lav2_Operador_PLC" : Int AT 4x403154, 2 s
      on ChangeValue: "S304_ActualizarOpEnPrincipal"(1)
   "Lav2_AlarmaVibracion" : Bit AT 0x3390, 2 s
      on ChangeValue: "SA1_email_Vibr"(); "S41_Write_Fall2BDD"()
   "Lav2_EnCiclo" : Bit AT 0x3081, 1 s
      on ChangeValue: "SA3_Act_HoraFinEstPrincLav2"()
   "Lav2_CicloFinalizado" : Bit AT 0x3251, 1 s
   "Lav2_Ciclograbado" : Bit AT 0x3231, 1 s
   "Lav2_ComienzoCiclo" : Bit AT 0x3230, 1 s
   "Lav2_Falla" : Int AT 4x403183, 500 ms
   "Lav2_ConfFalla" : Bit AT 0x3252, 1 s
   "Lav2_PulsParadaPres" : Bit AT 0x3253, 1 s
      on ChangeValue: "S41_Write_Fall2BDD"()
   "Lav2_Cli_0_Str" : WString[64], internal
   "Lav2_Cli_1_Str" : WString[64], internal
   "Lav2_Cli_2_Str" : WString[64], internal
   "Lav2_FinEstimado_Panel" : DateTime, internal
   "Lav2_ProgAGrabar" : Int AT 4x401025, 2 s
   "Lav2_Cont_IntentosGrabado" : Int, internal
   "Lav2_X0_iPres_SinAire" : Bit AT 0x2049, 1 s
   "Lav2_X1_iPres_Freno" : Bit AT 0x2050, 1 s
   "Lav2_X2_iTermico" : Bit AT 0x2051, 1 s
   "Lav2_X3_iSns_PCarga" : Bit AT 0x2052, 1 s
   "Lav2_X4_iSns_PDesc" : Bit AT 0x2053, 1 s
   "Lav2_X5_iPuls_DestrPuerta" : Bit AT 0x2054, 1 s
   "Lav2_X6_iSwitch_Vibra" : Bit AT 0x2055, 1 s
   "Lav2_X7_iFallVar" : Bit AT 0x2056, 1 s
   "Lav2_X11_iPulsMarcha" : Bit AT 0x2058, 1 s
   "Lav2_X12_iPulsPausa" : Bit AT 0x2059, 1 s
   "Lav2_X13_iNivBajo" : Bit AT 0x2060, 1 s
   "Lav2_X14_iBuscPtaCargArr" : Bit AT 0x2061, 1 s
   "Lav2_X15_iBuscPtaCargAba" : Bit AT 0x2062, 1 s
   "Lav2_X16_iBuscPtaDescArr" : Bit AT 0x2063, 1 s
   "Lav2_X17_iBuscPtaDescAba" : Bit AT 0x2064, 1 s
   "Lav2_X20_BloqMarchDesc" : Bit AT 0x2065, 1 s
   "Lav2_X21_iNiv_Alto" : Bit AT 0x2066, 1 s
   "Lav2_X22_iSns_Ind" : Bit AT 0x2067, 1 s
   "Lav2_X23_iPE" : Bit AT 0x2068, 1 s
   "Lav2_Y100_MachineOn" : Bit AT 1x102113, 1 s
   "Lav2_Y101_DosifPreLav" : Bit AT 1x102114, 1 s
   "Lav2_Y102_AvEjFinalNro2" : Bit AT 1x102115, 1 s
   "Lav2_Y103_AvEjFinalNro3" : Bit AT 1x102116, 1 s
   "Lav2_Y104_AvDosifLavNro1" : Bit AT 1x102117, 1 s
   "Lav2_Y105_Cloro_AvDosifL2" : Bit AT 1x102118, 1 s
   "Lav2_St_EnjIni" : Bit AT 0x3122, 1 s
   "Lav2_St_PrimLAv" : Bit AT 0x3127, 1 s
   "Lav2_St_EnjFin" : Bit AT 0x3131, 1 s
   "Lav2_St_EspCentr" : Bit AT 0x3133, 1 s
   "Lav2_St_Centr" : Bit AT 0x3134, 1 s
   "Lav2_St_FrenoMaquina" : Bit AT 0x3135, 1 s
   "Lav2_St_SegLav" : Bit AT 0x3138, 1 s
   "Lav2_St_PreLav" : Bit AT 0x3125, 1 s
   "Lav2_Programa_Anterior" : Int, internal
   "Lav2_grabFalla" : Bit AT 0x3253, 1 s
      on ChangeValue: "S41_Write_Fall2BDD"()
   "Lav2_CicloValido_CN" : Bit AT 0x3209, 1 s
   "Lav2_St_Ciclo" : Int AT 4x403182, 1 s
   "Lav2_FchFll_Ano" : Int AT 4x403198, 1 s
   "Lav2_FchFll_Mes" : Int AT 4x403197, 1 s
   "Lav2_FchFll_Dia" : Int AT 4x403196, 1 s
   "Lav2_FchFll_Hr" : Int AT 4x403195, 1 s
   "Lav2_FchFll_Mins" : Int AT 4x403194, 1 s
   "Lav2_FchFll_segs" : Int AT 4x403193, 1 s

HMI tags "Lavadora3"
   "Lav3_Programa" : Int AT 4x403158, 2 s
   "Lav3_Operador" : Int AT 4x403155, 2 s
      on ChangeValue: "S304_ActualizarOpEnPrincipal"(3)
   "Lav3_GrabarBDD" : Bit AT 0x3249, 2 s
      on ChangeValue: "S16_Write_data_Lav3"()
   "Lav3_CantRopa" : Int AT 4x403157, 2 s
   "Lav3_Alarma" : Bit AT 0x2057, 2 s
   "Lav3_FchFin_Ano" : Int AT 4x403172, 500 ms
   "Lav3_FchFin_Mes" : Int AT 4x403171, 500 ms
   "Lav3_FchFin_Dia" : Int AT 4x403170, 500 ms
   "Lav3_FchFin_Hr" : Int AT 4x403169, 500 ms
   "Lav3_FchFin_Min" : Int AT 4x403168, 500 ms
   "Lav3_FchFin_Seg" : Int AT 4x403167, 500 ms
   "Lav3_FchIni_Ano" : Int AT 4x403166, 1 s
   "Lav3_FchIni_Mes" : Int AT 4x403165, 1 s
   "Lav3_FchIni_Dia" : Int AT 4x403164, 1 s
   "Lav3_FchIni_Hr" : Int AT 4x403163, 1 s
   "Lav3_FchIni_Min" : Int AT 4x403162, 1 s
   "Lav3_FchIni_Seg" : Int AT 4x403161, 1 s
   "Lav3_Cliente_0" : Int AT 4x403160, 2 s
      on ChangeValue: "S104_ActualizarCliEmPrincipal"(3, 0)
   "Lav3_CicloValido" : Bit AT 0x3208, 100 ms
   "Lav3_Operador_Str" : WString[64], internal
   "Lav3_Fch_segs" : Int AT 4x404087, 500 ms
   "Lav3_Cliente_1" : Int AT 4x403174, 2 s
      on ChangeValue: "S104_ActualizarCliEmPrincipal"(3, 1)
   "Lav3_Cliente_2" : Int AT 4x403176, 2 s
      on ChangeValue: "S104_ActualizarCliEmPrincipal"(3, 2)
   "Lav3_Fch_Mins" : Int AT 4x404088, 500 ms
   "Lav3_Fch_Hr" : Int AT 4x404089, 500 ms
   "Lav3_Fch_Dia" : Int AT 4x404091, 500 ms
   "Lav3_Fch_Mes" : Int AT 4x404092, 500 ms
   "Lav3_Fch_Ano" : Int AT 4x404093, 500 ms
   "Lav3_Cliente_0_PLC" : Int AT 4x403159, 2 s
   "Lav3_Cliente_1_PLC" : Int AT 4x403173, 2 s
   "Lav3_Cliente_2_PLC" : Int AT 4x403175, 2 s
   "Lav3_Operador_PLC" : Int AT 4x403154, 2 s
      on ChangeValue: "S304_ActualizarOpEnPrincipal"(3)
   "Lav3_CantRopa_PLC" : Int AT 4x403156, 2 s
   "Lav3_AlarmaVibracion" : Bit AT 0x3390, 2 s
      on ChangeValue: "SA1_email_Vibr"(); "S42_Write_Fall3BDD"()
   "Lav3_EnCiclo" : Bit AT 0x3081, 1 s
      on ChangeValue: "SA3_Act_HoraFinEstPrincLav3"()
   "Lav3_CicloFinalizado" : Bit AT 0x3251, 1 s
   "Lav3_Ciclograbado" : Bit AT 0x3231, 1 s
   "Lav3_ComienzoCiclo" : Bit AT 0x3230, 1 s
   "Lav3_Falla" : Int AT 4x403183, 500 ms
   "Lav3_ConfFalla" : Bit AT 0x3252, 1 s
   "Lav3_PulsParadaPres" : Bit AT 0x3253, 1 s
      on ChangeValue: "S42_Write_Fall3BDD"()
   "Lav3_Cli_0_Str" : WString[64], internal
   "Lav3_Cli_1_Str" : WString[64], internal
   "Lav3_Cli_2_Str" : WString[64], internal
   "Lav3_FinEstimado_Panel" : DateTime, internal
   "Lav3_ProgAGrabar" : Int AT 4x401025, 2 s
   "Lav3_Cont_IntentosGrabado" : Int, internal
   "Lav3_X0_iPres_SinAire" : Bit AT 0x2049, 1 s
   "Lav3_X1_iPres_Freno" : Bit AT 0x2050, 1 s
   "Lav3_X2_iTermico" : Bit AT 0x2051, 1 s
   "Lav3_X3_iSns_PCarga" : Bit AT 0x2052, 1 s
   "Lav3_X4_iSns_PDesc" : Bit AT 0x2053, 1 s
   "Lav3_X5_iPuls_DestrPuerta" : Bit AT 0x2054, 1 s
   "Lav3_X6_iSwitch_Vibra" : Bit AT 0x2055, 1 s
   "Lav3_X7_iFallVar" : Bit AT 0x2056, 1 s
   "Lav3_X11_iPulsMarcha" : Bit AT 0x2058, 1 s
   "Lav3_X12_iPulsPausa" : Bit AT 0x2059, 1 s
   "Lav3_X13_iNivBajo" : Bit AT 0x2060, 1 s
   "Lav3_X14_iBuscPtaCargArr" : Bit AT 0x2061, 1 s
   "Lav3_X15_iBuscPtaCargAba" : Bit AT 0x2062, 1 s
   "Lav3_X16_iBuscPtaDescArr" : Bit AT 0x2063, 1 s
   "Lav3_X17_iBuscPtaDescAba" : Bit AT 0x2064, 1 s
   "Lav3_X20_BloqMarchDesc" : Bit AT 0x2065, 1 s
   "Lav3_X21_iNiv_Alto" : Bit AT 0x2066, 1 s
   "Lav3_X22_iSns_Ind" : Bit AT 0x2067, 1 s
   "Lav3_X23_iPE" : Bit AT 0x2068, 1 s
   "Lav3_Y100_MachineOn" : Bit AT 1x102113, 1 s
   "Lav3_Y101_DosifPreLav" : Bit AT 1x102114, 1 s
   "Lav3_Y102_AvEjFinalNro2" : Bit AT 1x102115, 1 s
   "Lav3_Y103_AvEjFinalNro3" : Bit AT 1x102116, 1 s
   "Lav3_Y104_AvDosifLavNro1" : Bit AT 1x102117, 1 s
   "Lav3_Y105_Cloro_AvDosifL2" : Bit AT 1x102118, 1 s
   "Lav3_St_EnjIni" : Bit AT 0x3122, 1 s
   "Lav3_St_PrimLAv" : Bit AT 0x3127, 1 s
   "Lav3_St_EnjFin" : Bit AT 0x3131, 1 s
   "Lav3_St_EspCentr" : Bit AT 0x3133, 1 s
   "Lav3_St_Centr" : Bit AT 0x3134, 1 s
   "Lav3_St_FrenoMaquina" : Bit AT 0x3135, 1 s
   "Lav3_St_SegLav" : Bit AT 0x3138, 1 s
   "Lav3_St_PreLav" : Bit AT 0x3125, 1 s
   "Lav3_Programa_Anterior" : Int, internal
   "Lav3_grabFalla" : Bit AT 0x3253, 1 s
      on ChangeValue: "S42_Write_Fall3BDD"()
   "Lav3_CicloValido_CN" : Bit AT 0x3209, 1 s
   "Lav3_St_Ciclo" : Int AT 4x403182, 1 s
   "Lav3_FchFll_Ano" : Int AT 4x403198, 1 s
   "Lav3_FchFll_Mes" : Int AT 4x403197, 1 s
   "Lav3_FchFll_Dia" : Int AT 4x403196, 1 s
   "Lav3_FchFll_Hr" : Int AT 4x403195, 1 s
   "Lav3_FchFll_Mins" : Int AT 4x403194, 1 s
   "Lav3_FchFll_segs" : Int AT 4x403193, 1 s

HMI tags "Supervisores"
   "Supervisor_Name_1" : WString[32], internal
   "Supervisor_Name_2" : WString[32], internal
   "Supervisor_Name_3" : WString[32], internal
   "Supervisor_Name_4" : WString[32], internal
   "Supervisor_ID_Camb" : Int, internal
   "Supervisor_Camb" : WString[10], internal
   "Supervisor_Actual_Ahora" : Bool = PLC HMI_Supervisor_Actual AT %M50.0, 1 s
      on ChangeValue: "S202_ActualizarSup_HMI"()
   "Supervisor_Name_Ahora" : WString[10] AT %DB1.DBX0.0

HMI tags "ListaOperadores"
   "ID_OP_1" : Int, internal
   "ID_OP_2" : Int, internal
   "ID_OP_3" : Int, internal
   "ID_OP_4" : Int, internal
   "ID_OP_5" : Int, internal
   "Name_OP_1" : WString[64], internal
   "Name_OP_2" : WString[64], internal
   "Name_OP_3" : WString[64], internal
   "Name_OP_4" : WString[64], internal
   "Name_OP_5" : WString[64], internal
   "ID_OP_Cambiar" : Int, internal
   "Name_OP_Cambiar" : WString[64], internal
   "ID_OP_Nuevo" : Int, internal
   "Name_OP_Nuevo" : WString[64], internal
   "OP_ID" : Int AT %DB1.DBW0
   "OP_Name" : WString[254] AT %DB1.DBX0.0

HMI tags "Lavadora4"
   "Lav4_Programa" : Int AT 4x403158, 2 s
   "Lav4_Operador" : Int AT 4x403155, 2 s
      on ChangeValue: "S304_ActualizarOpEnPrincipal"(4)
   "Lav4_GrabarBDD" : Bit AT 0x3244, 2 s
      on ChangeValue: "S18_Write_data_Lav4"()
   "Lav4_CantRopa" : Int AT 4x403157, 2 s
   "Lav4_Alarma" : Bit AT 0x2057, 2 s
   "Lav4_FchFin_Ano" : Int AT 4x403172, 500 ms
   "Lav4_FchFin_Mes" : Int AT 4x403171, 500 ms
   "Lav4_FchFin_Dia" : Int AT 4x403170, 500 ms
   "Lav4_FchFin_Hr" : Int AT 4x403169, 500 ms
   "Lav4_FchFin_Min" : Int AT 4x403168, 500 ms
   "Lav4_FchFin_Seg" : Int AT 4x403167, 500 ms
   "Lav4_FchIni_Ano" : Int AT 4x403166, 1 s
   "Lav4_FchIni_Mes" : Int AT 4x403165, 1 s
   "Lav4_FchIni_Dia" : Int AT 4x403164, 1 s
   "Lav4_FchIni_Hr" : Int AT 4x403163, 1 s
   "Lav4_FchIni_Min" : Int AT 4x403162, 1 s
   "Lav4_FchIni_Seg" : Int AT 4x403161, 1 s
   "Lav4_Cliente_0" : Int AT 4x403160, 2 s
      on ChangeValue: "S104_ActualizarCliEmPrincipal"(4, 0)
   "Lav4_CicloValido" : Bit AT 0x3208, 100 ms
   "Lav4_Operador_Str" : WString[64], internal
   "Lav4_Fch_segs" : Int AT 4x404087, 500 ms
   "Lav4_Cliente_1" : Int AT 4x403174, 2 s
      on ChangeValue: "S104_ActualizarCliEmPrincipal"(4, 1)
   "Lav4_Cliente_2" : Int AT 4x403176, 2 s
      on ChangeValue: "S104_ActualizarCliEmPrincipal"(4, 2)
   "Lav4_Fch_Mins" : Int AT 4x404088, 500 ms
   "Lav4_Fch_Hr" : Int AT 4x404089, 500 ms
   "Lav4_Fch_Dia" : Int AT 4x404091, 500 ms
   "Lav4_Fch_Mes" : Int AT 4x404092, 500 ms
   "Lav4_Fch_Ano" : Int AT 4x404093, 500 ms
   "Lav4_Cliente_0_PLC" : Int AT 4x403159, 2 s
   "Lav4_Cliente_1_PLC" : Int AT 4x403173, 2 s
   "Lav4_Cliente_2_PLC" : Int AT 4x403175, 2 s
   "Lav4_Operador_PLC" : Int AT 4x403154, 2 s
   "Lav4_CantRopa_PLC" : Int AT 4x403156, 2 s
   "Lav4_AlarmaVibracion" : Bit AT 0x3390, 2 s
      on ChangeValue: "SA1_email_Vibr"(); "S43_Write_Fall4BDD"()
   "Lav4_EnCiclo" : Bit AT 0x3081, 1 s
      on ChangeValue: "SA3_Act_HoraFinEstPrincLav4"()
   "Lav4_CicloFinalizado" : Bit AT 0x3251, 1 s
   "Lav4_Ciclograbado" : Bit AT 0x3231, 1 s
   "Lav4_ComienzoCiclo" : Bit AT 0x3230, 1 s
   "Lav4_Falla" : Int AT 4x403183, 500 ms
   "Lav4_ConfFalla" : Bit AT 0x3252, 1 s
   "Lav4_PulsParadaPres" : Bit AT 0x3253, 1 s
      on ChangeValue: "S43_Write_Fall4BDD"()
   "Lav4_Cli_0_Str" : WString[64], internal
   "Lav4_Cli_1_Str" : WString[64], internal
   "Lav4_Cli_2_Str" : WString[64], internal
   "Lav4_FinEstimado_Panel" : DateTime, internal
   "Lav4_Falla_Ant" : Int, internal
   "Lav4_ProgAGrabar" : Int AT 4x401025, 2 s
   "Lav4_Cont_IntentosGrabado" : Int, internal
   "Lav4_MachineOn" : Bit AT 1x102113, 1 s
   "Lav4_X0_iPres_SinAire" : Bit AT 0x2049, 1 s
   "Lav4_X1_iPres_Freno" : Bit AT 0x2050, 1 s
   "Lav4_X2_iTermico" : Bit AT 0x2051, 1 s
   "Lav4_X3_iSns_PCarga" : Bit AT 0x2052, 1 s
   "Lav4_X4_iSns_PDesc" : Bit AT 0x2053, 1 s
   "Lav4_X5_iPuls_DestrPuerta" : Bit AT 0x2054, 1 s
   "Lav4_X6_iSwitch_Vibra" : Bit AT 0x2055, 1 s
   "Lav4_X7_iFallVar" : Bit AT 0x2056, 1 s
   "Lav4_X11_iPulsMarcha" : Bit AT 0x2058, 1 s
   "Lav4_X12_iPulsPausa" : Bit AT 0x2059, 1 s
   "Lav4_X13_iNivBajo" : Bit AT 0x2060, 1 s
   "Lav4_X14_iBuscPtaCargArr" : Bit AT 0x2061, 1 s
   "Lav4_X15_iBuscPtaCargAba" : Bit AT 0x2062, 1 s
   "Lav4_X16_iBuscPtaDescArr" : Bit AT 0x2063, 1 s
   "Lav4_X17_iBuscPtaDescAba" : Bit AT 0x2064, 1 s
   "Lav4_X20_BloqMarchDesc" : Bit AT 0x2065, 1 s
   "Lav4_X21_iNiv_Alto" : Bit AT 0x2066, 1 s
   "Lav4_X22_iSns_Ind" : Bit AT 0x2067, 1 s
   "Lav4_X23_iPE" : Bit AT 0x2068, 1 s
   "Lav4_Y100_MachineOn" : Bit AT 1x102113, 1 s
   "Lav4_Y101_DosifPreLav" : Bit AT 1x102114, 1 s
   "Lav4_Y102_AvEjFinalNro2" : Bit AT 1x102115, 1 s
   "Lav4_Y103_AvEjFinalNro3" : Bit AT 1x102116, 1 s
   "Lav4_Y104_AvDosifLavNro1" : Bit AT 1x102117, 1 s
   "Lav4_Y105_Cloro_AvDosifL2" : Bit AT 1x102118, 1 s
   "Lav4_St_EnjIni" : Bit AT 0x3122, 1 s
   "Lav4_St_PrimLAv" : Bit AT 0x3127, 1 s
   "Lav4_St_EnjFin" : Bit AT 0x3131, 1 s
   "Lav4_St_EspCentr" : Bit AT 0x3133, 1 s
   "Lav4_St_Centr" : Bit AT 0x3134, 1 s
   "Lav4_St_FrenoMaquina" : Bit AT 0x3135, 1 s
   "Lav4_St_SegLav" : Bit AT 0x3138, 1 s
   "Lav4_St_PreLav" : Bit AT 0x3125, 1 s
   "Lav4_Programa_Anterior" : Int, internal
   "Lav4_grabFalla" : Bit AT 0x3253, 1 s
      on ChangeValue: "S43_Write_Fall4BDD"()
   "Lav4_CicloValido_CN" : Bit AT 0x3210, 1 s
   "Lav4_St_Ciclo" : Int AT 4x403182, 1 s
   "Lav4_Tiempo_Centrif" : Int AT 4x403087, 1 s
   "Lav4_FchFll_Ano" : Int AT 4x403198, 1 s
   "Lav4_FchFll_Mes" : Int AT 4x403197, 1 s
   "Lav4_FchFll_Dia" : Int AT 4x403196, 1 s
   "Lav4_FchFll_Hr" : Int AT 4x403195, 1 s
   "Lav4_FchFll_Mins" : Int AT 4x403194, 1 s
   "Lav4_FchFll_segs" : Int AT 4x403193, 1 s

HMI tags "ProLav4"
   "Lav4_Prog1_EnjIni_Cant" : Int AT 4x402562, 10 min
   "Lav4_Prog1_EnjIni_NivAg" : Int AT 4x402563, 10 min
   "Lav4_Prog1_EnjIni_Tiempo" : Int AT 4x402564, 10 min
   "Lav4_Prog1_PreLav_NivAg" : Int AT 4x402566, 10 min
   "Lav4_Prog1_PreLav_AgCaliente" : Int AT 4x402567, 10 min
   "Lav4_Prog1_Lav1_NivAg" : Int AT 4x402569, 10 min
   "Lav4_Prog1_Lav1_AgCaliente" : Int AT 4x402570, 10 min
   "Lav4_Prog1_EnjFin_Cant" : Int AT 4x402571, 10 min
   "Lav4_Prog1_Lav2_Tiempo" : Int AT 4x402617, 10 min
   "Lav4_Prog1_Lav2_NivAg" : Int AT 4x402572, 10 min
   "Lav4_Prog1_EnjFin_Tiempo" : Int AT 4x402573, 10 min
   "Lav4_Prog1_Lav2_AgCaliente" : Int AT 4x402574, 10 min
   "Lav4_Prog1_Centr_Tiempo" : Int AT 4x403092, 10 min
   "Lav4_Prog1_PreLav_Vapor" : Int AT 4x402576, 10 min
   "Lav4_Prog1_PreLav_Temperatura" : Int AT 4x402589, 10 min
   "Lav4_Prog1_Lav1_Temperatura" : Int AT 4x402591, 10 min
   "Lav4_Prog1_Lav2_Temperatura" : Int AT 4x401057, 10 min
   "Lav4_Prog1_PreLav_Tiempo" : Int AT 4x402565, 10 min
   "Lav4_Prog1_Lav1_Tiempo" : Int AT 4x402568, 10 min
   "Lav4_Prog2_EnjIni_Cant" : Int AT 4x402626, 10 min
   "Lav4_Prog2_EnjIni_NivAg" : Int AT 4x402627, 10 min
   "Lav4_Prog2_EnjIni_Tiempo" : Int AT 4x402628, 10 min
   "Lav4_Prog2_PreLav_NivAg" : Int AT 4x402630, 10 min
   "Lav4_Prog2_PreLav_AgCaliente" : Int AT 4x402631, 10 min
   "Lav4_Prog2_Lav1_NivAg" : Int AT 4x402633, 10 min
   "Lav4_Prog2_Lav1_AgCaliente" : Int AT 4x402634, 10 min
   "Lav4_Prog2_EnjFin_Cant" : Int AT 4x402635, 10 min
   "Lav4_Prog2_Lav2_Tiempo" : Int AT 4x402618, 10 min
   "Lav4_Prog2_Lav2_NivAg" : Int AT 4x402636, 10 min
   "Lav4_Prog2_EnjFin_Tiempo" : Int AT 4x402637, 10 min
   "Lav4_Prog2_Lav2_AgCaliente" : Int AT 4x402638, 10 min
   "Lav4_Prog2_Centr_Tiempo" : Int AT 4x403092, 10 min
   "Lav4_Prog2_PreLav_Vapor" : Int AT 4x402577, 10 min
   "Lav4_Prog2_PreLav_Temperatura" : Int AT 4x402592, 10 min
   "Lav4_Prog2_Lav1_Temperatura" : Int AT 4x402593, 10 min
   "Lav4_Prog2_Lav2_Temperatura" : Int AT 4x401058, 10 min
   "Lav4_Prog2_PreLav_Tiempo" : Int AT 4x402629, 10 min
   "Lav4_Prog2_Lav1_Tiempo" : Int AT 4x402632, 10 min
   "Lav4_Prog3_EnjIni_Cant" : Int AT 4x402690, 10 min
   "Lav4_Prog3_EnjIni_NivAg" : Int AT 4x402691, 10 min
   "Lav4_Prog3_EnjIni_Tiempo" : Int AT 4x402692, 10 min
   "Lav4_Prog3_PreLav_NivAg" : Int AT 4x402694, 10 min
   "Lav4_Prog3_PreLav_AgCaliente" : Int AT 4x402695, 10 min
   "Lav4_Prog3_Lav1_NivAg" : Int AT 4x402697, 10 min
   "Lav4_Prog3_Lav1_AgCaliente" : Int AT 4x402698, 10 min
   "Lav4_Prog3_EnjFin_Cant" : Int AT 4x402699, 10 min
   "Lav4_Prog3_Lav2_Tiempo" : Int AT 4x402619, 10 min
   "Lav4_Prog3_Lav2_NivAg" : Int AT 4x402700, 10 min
   "Lav4_Prog3_EnjFin_Tiempo" : Int AT 4x402701, 10 min
   "Lav4_Prog3_Lav2_AgCaliente" : Int AT 4x402702, 10 min
   "Lav4_Prog3_Centr_Tiempo" : Int AT 4x403092, 10 min
   "Lav4_Prog3_PreLav_Vapor" : Int AT 4x402579, 10 min
   "Lav4_Prog3_PreLav_Temperatura" : Int AT 4x402595, 10 min
   "Lav4_Prog3_Lav1_Temperatura" : Int AT 4x402597, 10 min
   "Lav4_Prog3_Lav2_Temperatura" : Int AT 4x401059, 10 min
   "Lav4_Prog3_PreLav_Tiempo" : Int AT 4x402693, 10 min
   "Lav4_Prog3_Lav1_Tiempo" : Int AT 4x402696, 10 min
   "Lav4_Prog4_EnjIni_Cant" : Int AT 4x402754, 10 min
   "Lav4_Prog4_EnjIni_NivAg" : Int AT 4x402755, 10 min
   "Lav4_Prog4_EnjIni_Tiempo" : Int AT 4x402756, 10 min
   "Lav4_Prog4_PreLav_NivAg" : Int AT 4x402758, 10 min
   "Lav4_Prog4_PreLav_AgCaliente" : Int AT 4x402759, 10 min
   "Lav4_Prog4_Lav1_NivAg" : Int AT 4x402761, 10 min
   "Lav4_Prog4_Lav1_AgCaliente" : Int AT 4x402762, 10 min
   "Lav4_Prog4_EnjFin_Cant" : Int AT 4x402763, 10 min
   "Lav4_Prog4_Lav2_Tiempo" : Int AT 4x402620, 10 min
   "Lav4_Prog4_Lav2_NivAg" : Int AT 4x402764, 10 min
   "Lav4_Prog4_EnjFin_Tiempo" : Int AT 4x402765, 10 min
   "Lav4_Prog4_Lav2_AgCaliente" : Int AT 4x402766, 10 min
   "Lav4_Prog4_Centr_Tiempo" : Int AT 4x403092, 10 min
   "Lav4_Prog4_PreLav_Vapor" : Int AT 4x402581, 10 min
   "Lav4_Prog4_PreLav_Temperatura" : Int AT 4x402599, 10 min
   "Lav4_Prog4_Lav1_Temperatura" : Int AT 4x402600, 10 min
   "Lav4_Prog4_Lav2_Temperatura" : Int AT 4x401060, 10 min
   "Lav4_Prog4_PreLav_Tiempo" : Int AT 4x402757, 10 min
   "Lav4_Prog4_Lav1_Tiempo" : Int AT 4x402760, 10 min
   "Lav4_Prog5_EnjIni_Cant" : Int AT 4x402818, 10 min
   "Lav4_Prog5_EnjIni_NivAg" : Int AT 4x402819, 10 min
   "Lav4_Prog5_EnjIni_Tiempo" : Int AT 4x402820, 10 min
   "Lav4_Prog5_PreLav_NivAg" : Int AT 4x402822, 10 min
   "Lav4_Prog5_PreLav_AgCaliente" : Int AT 4x402823, 10 min
   "Lav4_Prog5_Lav1_NivAg" : Int AT 4x402825, 10 min
   "Lav4_Prog5_Lav1_AgCaliente" : Int AT 4x402826, 10 min
   "Lav4_Prog5_EnjFin_Cant" : Int AT 4x402827, 10 min
   "Lav4_Prog5_Lav2_Tiempo" : Int AT 4x402621, 10 min
   "Lav4_Prog5_Lav2_NivAg" : Int AT 4x402828, 10 min
   "Lav4_Prog5_EnjFin_Tiempo" : Int AT 4x402829, 10 min
   "Lav4_Prog5_Lav2_AgCaliente" : Int AT 4x402830, 10 min
   "Lav4_Prog5_Centr_Tiempo" : Int AT 4x403092, 10 min
   "Lav4_Prog5_PreLav_Vapor" : Int AT 4x402583, 10 min
   "Lav4_Prog5_PreLav_Temperatura" : Int AT 4x402601, 10 min
   "Lav4_Prog5_Lav1_Temperatura" : Int AT 4x402603, 10 min
   "Lav4_Prog5_Lav2_Temperatura" : Int AT 4x401061, 10 min
   "Lav4_Prog5_PreLav_Tiempo" : Int AT 4x402821, 10 min
   "Lav4_Prog5_Lav1_Tiempo" : Int AT 4x402824, 10 min
   "Lav4_Prog6_EnjIni_Cant" : Int AT 4x402882, 10 min
   "Lav4_Prog6_EnjIni_NivAg" : Int AT 4x402883, 10 min
   "Lav4_Prog6_EnjIni_Tiempo" : Int AT 4x402884, 10 min
   "Lav4_Prog6_PreLav_NivAg" : Int AT 4x402886, 10 min
   "Lav4_Prog6_PreLav_AgCaliente" : Int AT 4x402887, 10 min
   "Lav4_Prog6_Lav1_NivAg" : Int AT 4x402889, 10 min
   "Lav4_Prog6_Lav1_AgCaliente" : Int AT 4x402890, 10 min
   "Lav4_Prog6_EnjFin_Cant" : Int AT 4x402891, 10 min
   "Lav4_Prog6_Lav2_Tiempo" : Int AT 4x402622, 10 min
   "Lav4_Prog6_Lav2_NivAg" : Int AT 4x402892, 10 min
   "Lav4_Prog6_EnjFin_Tiempo" : Int AT 4x402893, 10 min
   "Lav4_Prog6_Lav2_AgCaliente" : Int AT 4x402894, 10 min
   "Lav4_Prog6_Centr_Tiempo" : Int AT 4x403092, 10 min
   "Lav4_Prog6_PreLav_Vapor" : Int AT 4x402585, 10 min
   "Lav4_Prog6_PreLav_Temperatura" : Int AT 4x402605, 10 min
   "Lav4_Prog6_Lav1_Temperatura" : Int AT 4x402607, 10 min
   "Lav4_Prog6_Lav2_Temperatura" : Int AT 4x401062, 10 min
   "Lav4_Prog6_PreLav_Tiempo" : Int AT 4x402885, 10 min
   "Lav4_Prog6_Lav1_Tiempo" : Int AT 4x402888, 10 min
   "Lav4_Prog7_EnjIni_Cant" : Int AT 4x402953, 10 min
   "Lav4_Prog7_EnjIni_NivAg" : Int AT 4x402955, 10 min
   "Lav4_Prog7_EnjIni_Tiempo" : Int AT 4x402956, 10 min
   "Lav4_Prog7_PreLav_NivAg" : Int AT 4x402958, 10 min
   "Lav4_Prog7_PreLav_AgCaliente" : Int AT 4x402959, 10 min
   "Lav4_Prog7_Lav1_NivAg" : Int AT 4x402961, 10 min
   "Lav4_Prog7_Lav1_AgCaliente" : Int AT 4x402962, 10 min
   "Lav4_Prog7_EnjFin_Cant" : Int AT 4x402964, 10 min
   "Lav4_Prog7_Lav2_Tiempo" : Int AT 4x402963, 10 min
   "Lav4_Prog7_Lav2_NivAg" : Int AT 4x402965, 10 min
   "Lav4_Prog7_EnjFin_Tiempo" : Int AT 4x402966, 10 min
   "Lav4_Prog7_Lav2_AgCaliente" : Int AT 4x402967, 10 min
   "Lav4_Prog7_Centr_Tiempo" : Int AT 4x403092, 10 min
   "Lav4_Prog7_PreLav_Vapor" : Int AT 4x402969, 10 min
   "Lav4_Prog7_PreLav_Temperatura" : Int AT 4x402970, 10 min
   "Lav4_Prog7_Lav1_Temperatura" : Int AT 4x402971, 10 min
   "Lav4_Prog7_Lav2_Temperatura" : Int AT 4x401121, 10 min
   "Lav4_Prog7_PreLav_Tiempo" : Int AT 4x402957, 10 min
   "Lav4_Prog7_Lav1_Tiempo" : Int AT 4x402960, 10 min
   "Lav4_Prog8_EnjIni_Cant" : Int AT 4x402978, 10 min
   "Lav4_Prog8_EnjIni_NivAg" : Int AT 4x402979, 10 min
   "Lav4_Prog8_EnjIni_Tiempo" : Int AT 4x402980, 10 min
   "Lav4_Prog8_PreLav_NivAg" : Int AT 4x402982, 10 min
   "Lav4_Prog8_PreLav_AgCaliente" : Int AT 4x402983, 10 min
   "Lav4_Prog8_Lav1_NivAg" : Int AT 4x402985, 10 min
   "Lav4_Prog8_Lav1_AgCaliente" : Int AT 4x402986, 10 min
   "Lav4_Prog8_EnjFin_Cant" : Int AT 4x402988, 10 min
   "Lav4_Prog8_Lav2_Tiempo" : Int AT 4x402987, 10 min
   "Lav4_Prog8_Lav2_NivAg" : Int AT 4x402989, 10 min
   "Lav4_Prog8_EnjFin_Tiempo" : Int AT 4x402990, 10 min
   "Lav4_Prog8_Lav2_AgCaliente" : Int AT 4x402991, 10 min
   "Lav4_Prog8_Centr_Tiempo" : Int AT 4x403092, 10 min
   "Lav4_Prog8_PreLav_Vapor" : Int AT 4x402993, 10 min
   "Lav4_Prog8_PreLav_Temperatura" : Int AT 4x402994, 10 min
   "Lav4_Prog8_Lav1_Temperatura" : Int AT 4x402995, 10 min
   "Lav4_Prog8_Lav2_Temperatura" : Int AT 4x401186, 10 min
   "Lav4_Prog8_PreLav_Tiempo" : Int AT 4x402981, 10 min
   "Lav4_Prog8_Lav1_Tiempo" : Int AT 4x402984, 10 min
   "Lav4_Prog9_EnjIni_Cant" : Int AT 4x402996, 10 min
   "Lav4_Prog9_EnjIni_NivAg" : Int AT 4x402997, 10 min
   "Lav4_Prog9_EnjIni_Tiempo" : Int AT 4x402998, 10 min
   "Lav4_Prog9_PreLav_NivAg" : Int AT 4x403000, 10 min
   "Lav4_Prog9_PreLav_AgCaliente" : Int AT 4x403001, 10 min
   "Lav4_Prog9_Lav1_NivAg" : Int AT 4x403003, 10 min
   "Lav4_Prog9_Lav1_AgCaliente" : Int AT 4x403004, 10 min
   "Lav4_Prog9_EnjFin_Cant" : Int AT 4x403006, 10 min
   "Lav4_Prog9_Lav2_Tiempo" : Int AT 4x403005, 10 min
   "Lav4_Prog9_Lav2_NivAg" : Int AT 4x403007, 10 min
   "Lav4_Prog9_EnjFin_Tiempo" : Int AT 4x403008, 10 min
   "Lav4_Prog9_Lav2_AgCaliente" : Int AT 4x403009, 10 min
   "Lav4_Prog9_Centr_Tiempo" : Int AT 4x403092, 10 min
   "Lav4_Prog9_PreLav_Vapor" : Int AT 4x403011, 10 min
   "Lav4_Prog9_PreLav_Temperatura" : Int AT 4x403012, 10 min
   "Lav4_Prog9_Lav1_Temperatura" : Int AT 4x403013, 10 min
   "Lav4_Prog9_Lav2_Temperatura" : Int AT 4x401251, 10 min
   "Lav4_Prog9_PreLav_Tiempo" : Int AT 4x402999, 10 min
   "Lav4_Prog9_Lav1_Tiempo" : Int AT 4x403002, 10 min
   "Lav4_Prog10_EnjIni_Cant" : Int AT 4x403014, 10 min
   "Lav4_Prog10_EnjIni_NivAg" : Int AT 4x403015, 10 min
   "Lav4_Prog10_EnjIni_Tiempo" : Int AT 4x403016, 10 min
   "Lav4_Prog10_PreLav_NivAg" : Int AT 4x403018, 10 min
   "Lav4_Prog10_PreLav_AgCaliente" : Int AT 4x403019, 10 min
   "Lav4_Prog10_Lav1_NivAg" : Int AT 4x403021, 10 min
   "Lav4_Prog10_Lav1_AgCaliente" : Int AT 4x403022, 10 min
   "Lav4_Prog10_EnjFin_Cant" : Int AT 4x403024, 10 min
   "Lav4_Prog10_Lav2_Tiempo" : Int AT 4x403023, 10 min
   "Lav4_Prog10_Lav2_NivAg" : Int AT 4x403025, 10 min
   "Lav4_Prog10_EnjFin_Tiempo" : Int AT 4x403026, 10 min
   "Lav4_Prog10_Lav2_AgCaliente" : Int AT 4x403027, 10 min
   "Lav4_Prog10_Centr_Tiempo" : Int AT 4x403092, 10 min
   "Lav4_Prog10_PreLav_Vapor" : Int AT 4x403029, 10 min
   "Lav4_Prog10_PreLav_Temperatura" : Int AT 4x403030, 10 min
   "Lav4_Prog10_Lav1_Temperatura" : Int AT 4x403031, 10 min
   "Lav4_Prog10_Lav2_Temperatura" : Int AT 4x401316, 10 min
   "Lav4_Prog10_PreLav_Tiempo" : Int AT 4x403017, 10 min
   "Lav4_Prog10_Lav1_Tiempo" : Int AT 4x403020, 10 min
   "Lav4_Prog11_EnjIni_Cant" : Int AT 4x403033, 10 min
   "Lav4_Prog11_EnjIni_NivAg" : Int AT 4x403034, 10 min
   "Lav4_Prog11_EnjIni_Tiempo" : Int AT 4x403035, 10 min
   "Lav4_Prog11_PreLav_NivAg" : Int AT 4x403037, 10 min
   "Lav4_Prog11_PreLav_AgCaliente" : Int AT 4x403038, 10 min
   "Lav4_Prog11_Lav1_NivAg" : Int AT 4x403040, 10 min
   "Lav4_Prog11_Lav1_AgCaliente" : Int AT 4x403041, 10 min
   "Lav4_Prog11_EnjFin_Cant" : Int AT 4x403043, 10 min
   "Lav4_Prog11_Lav2_Tiempo" : Int AT 4x403042, 10 min
   "Lav4_Prog11_Lav2_NivAg" : Int AT 4x403044, 10 min
   "Lav4_Prog11_EnjFin_Tiempo" : Int AT 4x403045, 10 min
   "Lav4_Prog11_Lav2_AgCaliente" : Int AT 4x403046, 10 min
   "Lav4_Prog11_Centr_Tiempo" : Int AT 4x403092, 10 min
   "Lav4_Prog11_PreLav_Vapor" : Int AT 4x403048, 10 min
   "Lav4_Prog11_PreLav_Temperatura" : Int AT 4x403049, 10 min
   "Lav4_Prog11_Lav1_Temperatura" : Int AT 4x403050, 10 min
   "Lav4_Prog11_Lav2_Temperatura" : Int AT 4x401381, 10 min
   "Lav4_Prog11_PreLav_Tiempo" : Int AT 4x403036, 10 min
   "Lav4_Prog11_Lav1_Tiempo" : Int AT 4x403039, 10 min
   "Lav4_Prog12_EnjIni_Cant" : Int AT 4x403051, 10 min
   "Lav4_Prog12_EnjIni_NivAg" : Int AT 4x403052, 10 min
   "Lav4_Prog12_EnjIni_Tiempo" : Int AT 4x403053, 10 min
   "Lav4_Prog12_PreLav_NivAg" : Int AT 4x403055, 10 min
   "Lav4_Prog12_PreLav_AgCaliente" : Int AT 4x403056, 10 min
   "Lav4_Prog12_Lav1_NivAg" : Int AT 4x403058, 10 min
   "Lav4_Prog12_Lav1_AgCaliente" : Int AT 4x403059, 10 min
   "Lav4_Prog12_EnjFin_Cant" : Int AT 4x403061, 10 min
   "Lav4_Prog12_Lav2_Tiempo" : Int AT 4x403060, 10 min
   "Lav4_Prog12_Lav2_NivAg" : Int AT 4x403062, 10 min
   "Lav4_Prog12_EnjFin_Tiempo" : Int AT 4x403063, 10 min
   "Lav4_Prog12_Lav2_AgCaliente" : Int AT 4x403064, 10 min
   "Lav4_Prog12_Centr_Tiempo" : Int AT 4x403092, 10 min
   "Lav4_Prog12_PreLav_Vapor" : Int AT 4x403066, 10 min
   "Lav4_Prog12_PreLav_Temperatura" : Int AT 4x403067, 10 min
   "Lav4_Prog12_Lav1_Temperatura" : Int AT 4x403068, 10 min
   "Lav4_Prog12_Lav2_Temperatura" : Int AT 4x401382, 10 min
   "Lav4_Prog12_PreLav_Tiempo" : Int AT 4x403054, 10 min
   "Lav4_Prog12_Lav1_Tiempo" : Int AT 4x403057, 10 min
   "Lav4_Prog13_EnjIni_Cant" : Int AT 4x402091, 10 min
   "Lav4_Prog13_EnjIni_NivAg" : Int AT 4x402092, 10 min
   "Lav4_Prog13_EnjIni_Tiempo" : Int AT 4x402093, 10 min
   "Lav4_Prog13_PreLav_NivAg" : Int AT 4x402095, 10 min
   "Lav4_Prog13_PreLav_AgCaliente" : Int AT 4x402096, 10 min
   "Lav4_Prog13_Lav1_NivAg" : Int AT 4x402098, 10 min
   "Lav4_Prog13_Lav1_AgCaliente" : Int AT 4x402099, 10 min
   "Lav4_Prog13_EnjFin_Cant" : Int AT 4x402101, 10 min
   "Lav4_Prog13_Lav2_Tiempo" : Int AT 4x402100, 10 min
   "Lav4_Prog13_Lav2_NivAg" : Int AT 4x402102, 10 min
   "Lav4_Prog13_EnjFin_Tiempo" : Int AT 4x402103, 10 min
   "Lav4_Prog13_Lav2_AgCaliente" : Int AT 4x402104, 10 min
   "Lav4_Prog13_Centr_Tiempo" : Int AT 4x403092, 10 min
   "Lav4_Prog13_PreLav_Vapor" : Int AT 4x402106, 10 min
   "Lav4_Prog13_PreLav_Temperatura" : Int AT 4x402107, 10 min
   "Lav4_Prog13_Lav1_Temperatura" : Int AT 4x402108, 10 min
   "Lav4_Prog13_Lav2_Temperatura" : Int AT 4x401383, 10 min
   "Lav4_Prog13_PreLav_Tiempo" : Int AT 4x402094, 10 min
   "Lav4_Prog13_Lav1_Tiempo" : Int AT 4x402097, 10 min
   "Lav4_Prog14_EnjIni_Cant" : Int AT 4x402155, 10 min
   "Lav4_Prog14_EnjIni_NivAg" : Int AT 4x402156, 10 min
   "Lav4_Prog14_EnjIni_Tiempo" : Int AT 4x402157, 10 min
   "Lav4_Prog14_PreLav_NivAg" : Int AT 4x402159, 10 min
   "Lav4_Prog14_PreLav_AgCaliente" : Int AT 4x402160, 10 min
   "Lav4_Prog14_Lav1_NivAg" : Int AT 4x402162, 10 min
   "Lav4_Prog14_Lav1_AgCaliente" : Int AT 4x402163, 10 min
   "Lav4_Prog14_EnjFin_Cant" : Int AT 4x402165, 10 min
   "Lav4_Prog14_Lav2_Tiempo" : Int AT 4x402164, 10 min
   "Lav4_Prog14_Lav2_NivAg" : Int AT 4x402166, 10 min
   "Lav4_Prog14_EnjFin_Tiempo" : Int AT 4x402167, 10 min
   "Lav4_Prog14_Lav2_AgCaliente" : Int AT 4x402168, 10 min
   "Lav4_Prog14_Centr_Tiempo" : Int AT 4x403092, 10 min
   "Lav4_Prog14_PreLav_Vapor" : Int AT 4x402170, 10 min
   "Lav4_Prog14_PreLav_Temperatura" : Int AT 4x402171, 10 min
   "Lav4_Prog14_Lav1_Temperatura" : Int AT 4x402172, 10 min
   "Lav4_Prog14_Lav2_Temperatura" : Int AT 4x401384, 10 min
   "Lav4_Prog14_PreLav_Tiempo" : Int AT 4x402158, 10 min
   "Lav4_Prog14_Lav1_Tiempo" : Int AT 4x402161, 10 min
   "Lav4_Prog15_EnjIni_Cant" : Int AT 4x402219, 10 min
   "Lav4_Prog15_EnjIni_NivAg" : Int AT 4x402220, 10 min
   "Lav4_Prog15_EnjIni_Tiempo" : Int AT 4x402221, 10 min
   "Lav4_Prog15_PreLav_NivAg" : Int AT 4x402223, 10 min
   "Lav4_Prog15_PreLav_AgCaliente" : Int AT 4x402224, 10 min
   "Lav4_Prog15_Lav1_NivAg" : Int AT 4x402226, 10 min
   "Lav4_Prog15_Lav1_AgCaliente" : Int AT 4x402227, 10 min
   "Lav4_Prog15_EnjFin_Cant" : Int AT 4x402229, 10 min
   "Lav4_Prog15_Lav2_Tiempo" : Int AT 4x402228, 10 min
   "Lav4_Prog15_Lav2_NivAg" : Int AT 4x402230, 10 min
   "Lav4_Prog15_EnjFin_Tiempo" : Int AT 4x402231, 10 min
   "Lav4_Prog15_Lav2_AgCaliente" : Int AT 4x402232, 10 min
   "Lav4_Prog15_Centr_Tiempo" : Int AT 4x403092, 10 min
   "Lav4_Prog15_PreLav_Vapor" : Int AT 4x402234, 10 min
   "Lav4_Prog15_PreLav_Temperatura" : Int AT 4x402235, 10 min
   "Lav4_Prog15_Lav1_Temperatura" : Int AT 4x402236, 10 min
   "Lav4_Prog15_Lav2_Temperatura" : Int AT 4x401385, 10 min
   "Lav4_Prog15_PreLav_Tiempo" : Int AT 4x402222, 10 min
   "Lav4_Prog15_Lav1_Tiempo" : Int AT 4x402225, 10 min

HMI tags "ProLav3"
   "Lav3_Prog1_EnjIni_Cant" : Int AT 4x402562, 10 min
   "Lav3_Prog1_EnjIni_NivAg" : Int AT 4x402563, 10 min
   "Lav3_Prog1_EnjIni_Tiempo" : Int AT 4x402564, 10 min
   "Lav3_Prog1_PreLav_NivAg" : Int AT 4x402566, 10 min
   "Lav3_Prog1_PreLav_AgCaliente" : Int AT 4x402567, 10 min
   "Lav3_Prog1_Lav1_NivAg" : Int AT 4x402569, 10 min
   "Lav3_Prog1_Lav1_AgCaliente" : Int AT 4x402570, 10 min
   "Lav3_Prog1_EnjFin_Cant" : Int AT 4x402571, 10 min
   "Lav3_Prog1_Lav2_Tiempo" : Int AT 4x402617, 10 min
   "Lav3_Prog1_Lav2_NivAg" : Int AT 4x402572, 10 min
   "Lav3_Prog1_EnjFin_Tiempo" : Int AT 4x402573, 10 min
   "Lav3_Prog1_Lav2_AgCaliente" : Int AT 4x402574, 10 min
   "Lav3_Prog1_Centr_Tiempo" : Int AT 4x402575, 10 min
   "Lav3_Prog1_PreLav_Vapor" : Int AT 4x402576, 10 min
   "Lav3_Prog1_PreLav_Temperatura" : Int AT 4x402589, 10 min
   "Lav3_Prog1_Lav1_Temperatura" : Int AT 4x402591, 10 min
   "Lav3_Prog1_Lav2_Temperatura" : Int AT 4x401057, 10 min
   "Lav3_Prog1_PreLav_Tiempo" : Int AT 4x402565, 10 min
   "Lav3_Prog1_Lav1_Tiempo" : Int AT 4x402568, 10 min
   "Lav3_Prog2_EnjIni_Cant" : Int AT 4x402626, 10 min
   "Lav3_Prog2_EnjIni_NivAg" : Int AT 4x402627, 10 min
   "Lav3_Prog2_EnjIni_Tiempo" : Int AT 4x402628, 10 min
   "Lav3_Prog2_PreLav_NivAg" : Int AT 4x402630, 10 min
   "Lav3_Prog2_PreLav_AgCaliente" : Int AT 4x402631, 10 min
   "Lav3_Prog2_Lav1_NivAg" : Int AT 4x402633, 10 min
   "Lav3_Prog2_Lav1_AgCaliente" : Int AT 4x402634, 10 min
   "Lav3_Prog2_EnjFin_Cant" : Int AT 4x402635, 10 min
   "Lav3_Prog2_Lav2_Tiempo" : Int AT 4x402618, 10 min
   "Lav3_Prog2_Lav2_NivAg" : Int AT 4x402636, 10 min
   "Lav3_Prog2_EnjFin_Tiempo" : Int AT 4x402637, 10 min
   "Lav3_Prog2_Lav2_AgCaliente" : Int AT 4x402638, 10 min
   "Lav3_Prog2_Centr_Tiempo" : Int AT 4x402639, 10 min
   "Lav3_Prog2_PreLav_Vapor" : Int AT 4x402577, 10 min
   "Lav3_Prog2_PreLav_Temperatura" : Int AT 4x402592, 10 min
   "Lav3_Prog2_Lav1_Temperatura" : Int AT 4x402593, 10 min
   "Lav3_Prog2_Lav2_Temperatura" : Int AT 4x401058, 10 min
   "Lav3_Prog2_PreLav_Tiempo" : Int AT 4x402629, 10 min
   "Lav3_Prog2_Lav1_Tiempo" : Int AT 4x402632, 10 min
   "Lav3_Prog3_EnjIni_Cant" : Int AT 4x402690, 10 min
   "Lav3_Prog3_EnjIni_NivAg" : Int AT 4x402691, 10 min
   "Lav3_Prog3_EnjIni_Tiempo" : Int AT 4x402692, 10 min
   "Lav3_Prog3_PreLav_NivAg" : Int AT 4x402694, 10 min
   "Lav3_Prog3_PreLav_AgCaliente" : Int AT 4x402695, 10 min
   "Lav3_Prog3_Lav1_NivAg" : Int AT 4x402697, 10 min
   "Lav3_Prog3_Lav1_AgCaliente" : Int AT 4x402698, 10 min
   "Lav3_Prog3_EnjFin_Cant" : Int AT 4x402699, 10 min
   "Lav3_Prog3_Lav2_Tiempo" : Int AT 4x402619, 10 min
   "Lav3_Prog3_Lav2_NivAg" : Int AT 4x402700, 10 min
   "Lav3_Prog3_EnjFin_Tiempo" : Int AT 4x402701, 10 min
   "Lav3_Prog3_Lav2_AgCaliente" : Int AT 4x402702, 10 min
   "Lav3_Prog3_Centr_Tiempo" : Int AT 4x402703, 10 min
   "Lav3_Prog3_PreLav_Vapor" : Int AT 4x402579, 10 min
   "Lav3_Prog3_PreLav_Temperatura" : Int AT 4x402595, 10 min
   "Lav3_Prog3_Lav1_Temperatura" : Int AT 4x402597, 10 min
   "Lav3_Prog3_Lav2_Temperatura" : Int AT 4x401059, 10 min
   "Lav3_Prog3_PreLav_Tiempo" : Int AT 4x402693, 10 min
   "Lav3_Prog3_Lav1_Tiempo" : Int AT 4x402696, 10 min
   "Lav3_Prog4_EnjIni_Cant" : Int AT 4x402754, 10 min
   "Lav3_Prog4_EnjIni_NivAg" : Int AT 4x402755, 10 min
   "Lav3_Prog4_EnjIni_Tiempo" : Int AT 4x402756, 10 min
   "Lav3_Prog4_PreLav_NivAg" : Int AT 4x402758, 10 min
   "Lav3_Prog4_PreLav_AgCaliente" : Int AT 4x402759, 10 min
   "Lav3_Prog4_Lav1_NivAg" : Int AT 4x402761, 10 min
   "Lav3_Prog4_Lav1_AgCaliente" : Int AT 4x402762, 10 min
   "Lav3_Prog4_EnjFin_Cant" : Int AT 4x402763, 10 min
   "Lav3_Prog4_Lav2_Tiempo" : Int AT 4x402620, 10 min
   "Lav3_Prog4_Lav2_NivAg" : Int AT 4x402764, 10 min
   "Lav3_Prog4_EnjFin_Tiempo" : Int AT 4x402765, 10 min
   "Lav3_Prog4_Lav2_AgCaliente" : Int AT 4x402766, 10 min
   "Lav3_Prog4_Centr_Tiempo" : Int AT 4x402767, 10 min
   "Lav3_Prog4_PreLav_Vapor" : Int AT 4x402581, 10 min
   "Lav3_Prog4_PreLav_Temperatura" : Int AT 4x402599, 10 min
   "Lav3_Prog4_Lav1_Temperatura" : Int AT 4x402600, 10 min
   "Lav3_Prog4_Lav2_Temperatura" : Int AT 4x401060, 10 min
   "Lav3_Prog4_PreLav_Tiempo" : Int AT 4x402757, 10 min
   "Lav3_Prog4_Lav1_Tiempo" : Int AT 4x402760, 10 min
   "Lav3_Prog5_EnjIni_Cant" : Int AT 4x402818, 10 min
   "Lav3_Prog5_EnjIni_NivAg" : Int AT 4x402819, 10 min
   "Lav3_Prog5_EnjIni_Tiempo" : Int AT 4x402820, 10 min
   "Lav3_Prog5_PreLav_NivAg" : Int AT 4x402822, 10 min
   "Lav3_Prog5_PreLav_AgCaliente" : Int AT 4x402823, 10 min
   "Lav3_Prog5_Lav1_NivAg" : Int AT 4x402825, 10 min
   "Lav3_Prog5_Lav1_AgCaliente" : Int AT 4x402826, 10 min
   "Lav3_Prog5_EnjFin_Cant" : Int AT 4x402827, 10 min
   "Lav3_Prog5_Lav2_Tiempo" : Int AT 4x402621, 10 min
   "Lav3_Prog5_Lav2_NivAg" : Int AT 4x402828, 10 min
   "Lav3_Prog5_EnjFin_Tiempo" : Int AT 4x402829, 10 min
   "Lav3_Prog5_Lav2_AgCaliente" : Int AT 4x402830, 10 min
   "Lav3_Prog5_Centr_Tiempo" : Int AT 4x402831, 10 min
   "Lav3_Prog5_PreLav_Vapor" : Int AT 4x402583, 10 min
   "Lav3_Prog5_PreLav_Temperatura" : Int AT 4x402601, 10 min
   "Lav3_Prog5_Lav1_Temperatura" : Int AT 4x402603, 10 min
   "Lav3_Prog5_Lav2_Temperatura" : Int AT 4x401061, 10 min
   "Lav3_Prog5_PreLav_Tiempo" : Int AT 4x402821, 10 min
   "Lav3_Prog5_Lav1_Tiempo" : Int AT 4x402824, 10 min
   "Lav3_Prog6_EnjIni_Cant" : Int AT 4x402882, 10 min
   "Lav3_Prog6_EnjIni_NivAg" : Int AT 4x402883, 10 min
   "Lav3_Prog6_EnjIni_Tiempo" : Int AT 4x402884, 10 min
   "Lav3_Prog6_PreLav_NivAg" : Int AT 4x402886, 10 min
   "Lav3_Prog6_PreLav_AgCaliente" : Int AT 4x402887, 10 min
   "Lav3_Prog6_Lav1_NivAg" : Int AT 4x402889, 10 min
   "Lav3_Prog6_Lav1_AgCaliente" : Int AT 4x402890, 10 min
   "Lav3_Prog6_EnjFin_Cant" : Int AT 4x402891, 10 min
   "Lav3_Prog6_Lav2_Tiempo" : Int AT 4x402622, 10 min
   "Lav3_Prog6_Lav2_NivAg" : Int AT 4x402892, 10 min
   "Lav3_Prog6_EnjFin_Tiempo" : Int AT 4x402893, 10 min
   "Lav3_Prog6_Lav2_AgCaliente" : Int AT 4x402894, 10 min
   "Lav3_Prog6_Centr_Tiempo" : Int AT 4x402895, 10 min
   "Lav3_Prog6_PreLav_Vapor" : Int AT 4x402585, 10 min
   "Lav3_Prog6_PreLav_Temperatura" : Int AT 4x402605, 10 min
   "Lav3_Prog6_Lav1_Temperatura" : Int AT 4x402607, 10 min
   "Lav3_Prog6_Lav2_Temperatura" : Int AT 4x401062, 10 min
   "Lav3_Prog6_PreLav_Tiempo" : Int AT 4x402885, 10 min
   "Lav3_Prog6_Lav1_Tiempo" : Int AT 4x402888, 10 min
   "Lav3_Prog7_EnjIni_Cant" : Int AT 4x402953, 10 min
   "Lav3_Prog7_EnjIni_NivAg" : Int AT 4x402955, 10 min
   "Lav3_Prog7_EnjIni_Tiempo" : Int AT 4x402956, 10 min
   "Lav3_Prog7_PreLav_NivAg" : Int AT 4x402958, 10 min
   "Lav3_Prog7_PreLav_AgCaliente" : Int AT 4x402959, 10 min
   "Lav3_Prog7_Lav1_NivAg" : Int AT 4x402961, 10 min
   "Lav3_Prog7_Lav1_AgCaliente" : Int AT 4x402962, 10 min
   "Lav3_Prog7_EnjFin_Cant" : Int AT 4x402964, 10 min
   "Lav3_Prog7_Lav2_Tiempo" : Int AT 4x402963, 10 min
   "Lav3_Prog7_Lav2_NivAg" : Int AT 4x402965, 10 min
   "Lav3_Prog7_EnjFin_Tiempo" : Int AT 4x402966, 10 min
   "Lav3_Prog7_Lav2_AgCaliente" : Int AT 4x402967, 10 min
   "Lav3_Prog7_Centr_Tiempo" : Int AT 4x402968, 10 min
   "Lav3_Prog7_PreLav_Vapor" : Int AT 4x402969, 10 min
   "Lav3_Prog7_PreLav_Temperatura" : Int AT 4x402970, 10 min
   "Lav3_Prog7_Lav1_Temperatura" : Int AT 4x402971, 10 min
   "Lav3_Prog7_Lav2_Temperatura" : Int AT 4x401121, 10 min
   "Lav3_Prog7_PreLav_Tiempo" : Int AT 4x402957, 10 min
   "Lav3_Prog7_Lav1_Tiempo" : Int AT 4x402960, 10 min
   "Lav3_Prog8_EnjIni_Cant" : Int AT 4x402978, 10 min
   "Lav3_Prog8_EnjIni_NivAg" : Int AT 4x402979, 10 min
   "Lav3_Prog8_EnjIni_Tiempo" : Int AT 4x402980, 10 min
   "Lav3_Prog8_PreLav_NivAg" : Int AT 4x402982, 10 min
   "Lav3_Prog8_PreLav_AgCaliente" : Int AT 4x402983, 10 min
   "Lav3_Prog8_Lav1_NivAg" : Int AT 4x402985, 10 min
   "Lav3_Prog8_Lav1_AgCaliente" : Int AT 4x402986, 10 min
   "Lav3_Prog8_EnjFin_Cant" : Int AT 4x402988, 10 min
   "Lav3_Prog8_Lav2_Tiempo" : Int AT 4x402987, 10 min
   "Lav3_Prog8_Lav2_NivAg" : Int AT 4x402989, 10 min
   "Lav3_Prog8_EnjFin_Tiempo" : Int AT 4x402990, 10 min
   "Lav3_Prog8_Lav2_AgCaliente" : Int AT 4x402991, 10 min
   "Lav3_Prog8_Centr_Tiempo" : Int AT 4x402992, 10 min
   "Lav3_Prog8_PreLav_Vapor" : Int AT 4x402993, 10 min
   "Lav3_Prog8_PreLav_Temperatura" : Int AT 4x402994, 10 min
   "Lav3_Prog8_Lav1_Temperatura" : Int AT 4x402995, 10 min
   "Lav3_Prog8_Lav2_Temperatura" : Int AT 4x401186, 10 min
   "Lav3_Prog8_PreLav_Tiempo" : Int AT 4x402981, 10 min
   "Lav3_Prog8_Lav1_Tiempo" : Int AT 4x402984, 10 min
   "Lav3_Prog9_EnjIni_Cant" : Int AT 4x402996, 10 min
   "Lav3_Prog9_EnjIni_NivAg" : Int AT 4x402997, 10 min
   "Lav3_Prog9_EnjIni_Tiempo" : Int AT 4x402998, 10 min
   "Lav3_Prog9_PreLav_NivAg" : Int AT 4x403000, 10 min
   "Lav3_Prog9_PreLav_AgCaliente" : Int AT 4x403001, 10 min
   "Lav3_Prog9_Lav1_NivAg" : Int AT 4x403003, 10 min
   "Lav3_Prog9_Lav1_AgCaliente" : Int AT 4x403004, 10 min
   "Lav3_Prog9_EnjFin_Cant" : Int AT 4x403006, 10 min
   "Lav3_Prog9_Lav2_Tiempo" : Int AT 4x403005, 10 min
   "Lav3_Prog9_Lav2_NivAg" : Int AT 4x403007, 10 min
   "Lav3_Prog9_EnjFin_Tiempo" : Int AT 4x403008, 10 min
   "Lav3_Prog9_Lav2_AgCaliente" : Int AT 4x403009, 10 min
   "Lav3_Prog9_Centr_Tiempo" : Int AT 4x403010, 10 min
   "Lav3_Prog9_PreLav_Vapor" : Int AT 4x403011, 10 min
   "Lav3_Prog9_PreLav_Temperatura" : Int AT 4x403012, 10 min
   "Lav3_Prog9_Lav1_Temperatura" : Int AT 4x403013, 10 min
   "Lav3_Prog9_Lav2_Temperatura" : Int AT 4x401251, 10 min
   "Lav3_Prog9_PreLav_Tiempo" : Int AT 4x402999, 10 min
   "Lav3_Prog9_Lav1_Tiempo" : Int AT 4x403002, 10 min
   "Lav3_Prog10_EnjIni_Cant" : Int AT 4x403014, 10 min
   "Lav3_Prog10_EnjIni_NivAg" : Int AT 4x403015, 10 min
   "Lav3_Prog10_EnjIni_Tiempo" : Int AT 4x403016, 10 min
   "Lav3_Prog10_PreLav_NivAg" : Int AT 4x403018, 10 min
   "Lav3_Prog10_PreLav_AgCaliente" : Int AT 4x403019, 10 min
   "Lav3_Prog10_Lav1_NivAg" : Int AT 4x403021, 10 min
   "Lav3_Prog10_Lav1_AgCaliente" : Int AT 4x403022, 10 min
   "Lav3_Prog10_EnjFin_Cant" : Int AT 4x403024, 10 min
   "Lav3_Prog10_Lav2_Tiempo" : Int AT 4x403023, 10 min
   "Lav3_Prog10_Lav2_NivAg" : Int AT 4x403025, 10 min
   "Lav3_Prog10_EnjFin_Tiempo" : Int AT 4x403026, 10 min
   "Lav3_Prog10_Lav2_AgCaliente" : Int AT 4x403027, 10 min
   "Lav3_Prog10_Centr_Tiempo" : Int AT 4x403028, 10 min
   "Lav3_Prog10_PreLav_Vapor" : Int AT 4x403029, 10 min
   "Lav3_Prog10_PreLav_Temperatura" : Int AT 4x403030, 10 min
   "Lav3_Prog10_Lav1_Temperatura" : Int AT 4x403031, 10 min
   "Lav3_Prog10_Lav2_Temperatura" : Int AT 4x401316, 10 min
   "Lav3_Prog10_PreLav_Tiempo" : Int AT 4x403017, 10 min
   "Lav3_Prog10_Lav1_Tiempo" : Int AT 4x403020, 10 min
   "Lav3_Prog11_EnjIni_Cant" : Int AT 4x403033, 10 min
   "Lav3_Prog11_EnjIni_NivAg" : Int AT 4x403034, 10 min
   "Lav3_Prog11_EnjIni_Tiempo" : Int AT 4x403035, 10 min
   "Lav3_Prog11_PreLav_NivAg" : Int AT 4x403037, 10 min
   "Lav3_Prog11_PreLav_AgCaliente" : Int AT 4x403038, 10 min
   "Lav3_Prog11_Lav1_NivAg" : Int AT 4x403040, 10 min
   "Lav3_Prog11_Lav1_AgCaliente" : Int AT 4x403041, 10 min
   "Lav3_Prog11_EnjFin_Cant" : Int AT 4x403043, 10 min
   "Lav3_Prog11_Lav2_Tiempo" : Int AT 4x403042, 10 min
   "Lav3_Prog11_Lav2_NivAg" : Int AT 4x403044, 10 min
   "Lav3_Prog11_EnjFin_Tiempo" : Int AT 4x403045, 10 min
   "Lav3_Prog11_Lav2_AgCaliente" : Int AT 4x403046, 10 min
   "Lav3_Prog11_Centr_Tiempo" : Int AT 4x403047, 10 min
   "Lav3_Prog11_PreLav_Vapor" : Int AT 4x403048, 10 min
   "Lav3_Prog11_PreLav_Temperatura" : Int AT 4x403049, 10 min
   "Lav3_Prog11_Lav1_Temperatura" : Int AT 4x403050, 10 min
   "Lav3_Prog11_Lav2_Temperatura" : Int AT 4x401381, 10 min
   "Lav3_Prog11_PreLav_Tiempo" : Int AT 4x403036, 10 min
   "Lav3_Prog11_Lav1_Tiempo" : Int AT 4x403039, 10 min
   "Lav3_Prog12_EnjIni_Cant" : Int AT 4x403051, 10 min
   "Lav3_Prog12_EnjIni_NivAg" : Int AT 4x403052, 10 min
   "Lav3_Prog12_EnjIni_Tiempo" : Int AT 4x403053, 10 min
   "Lav3_Prog12_PreLav_NivAg" : Int AT 4x403055, 10 min
   "Lav3_Prog12_PreLav_AgCaliente" : Int AT 4x403056, 10 min
   "Lav3_Prog12_Lav1_NivAg" : Int AT 4x403058, 10 min
   "Lav3_Prog12_Lav1_AgCaliente" : Int AT 4x403059, 10 min
   "Lav3_Prog12_EnjFin_Cant" : Int AT 4x403061, 10 min
   "Lav3_Prog12_Lav2_Tiempo" : Int AT 4x403060, 10 min
   "Lav3_Prog12_Lav2_NivAg" : Int AT 4x403062, 10 min
   "Lav3_Prog12_EnjFin_Tiempo" : Int AT 4x403063, 10 min
   "Lav3_Prog12_Lav2_AgCaliente" : Int AT 4x403064, 10 min
   "Lav3_Prog12_Centr_Tiempo" : Int AT 4x403065, 10 min
   "Lav3_Prog12_PreLav_Vapor" : Int AT 4x403066, 10 min
   "Lav3_Prog12_PreLav_Temperatura" : Int AT 4x403067, 10 min
   "Lav3_Prog12_Lav1_Temperatura" : Int AT 4x403068, 10 min
   "Lav3_Prog12_Lav2_Temperatura" : Int AT 4x401382, 10 min
   "Lav3_Prog12_PreLav_Tiempo" : Int AT 4x403054, 10 min
   "Lav3_Prog12_Lav1_Tiempo" : Int AT 4x403057, 10 min
   "Lav3_Prog13_EnjIni_Cant" : Int AT 4x402091, 10 min
   "Lav3_Prog13_EnjIni_NivAg" : Int AT 4x402092, 10 min
   "Lav3_Prog13_EnjIni_Tiempo" : Int AT 4x402093, 10 min
   "Lav3_Prog13_PreLav_NivAg" : Int AT 4x402095, 10 min
   "Lav3_Prog13_PreLav_AgCaliente" : Int AT 4x402096, 10 min
   "Lav3_Prog13_Lav1_NivAg" : Int AT 4x402098, 10 min
   "Lav3_Prog13_Lav1_AgCaliente" : Int AT 4x402099, 10 min
   "Lav3_Prog13_EnjFin_Cant" : Int AT 4x402101, 10 min
   "Lav3_Prog13_Lav2_Tiempo" : Int AT 4x402100, 10 min
   "Lav3_Prog13_Lav2_NivAg" : Int AT 4x402102, 10 min
   "Lav3_Prog13_EnjFin_Tiempo" : Int AT 4x402103, 10 min
   "Lav3_Prog13_Lav2_AgCaliente" : Int AT 4x402104, 10 min
   "Lav3_Prog13_Centr_Tiempo" : Int AT 4x402105, 10 min
   "Lav3_Prog13_PreLav_Vapor" : Int AT 4x402106, 10 min
   "Lav3_Prog13_PreLav_Temperatura" : Int AT 4x402107, 10 min
   "Lav3_Prog13_Lav1_Temperatura" : Int AT 4x402108, 10 min
   "Lav3_Prog13_Lav2_Temperatura" : Int AT 4x401383, 10 min
   "Lav3_Prog13_PreLav_Tiempo" : Int AT 4x402094, 10 min
   "Lav3_Prog13_Lav1_Tiempo" : Int AT 4x402097, 10 min
   "Lav3_Prog14_EnjIni_Cant" : Int AT 4x402155, 10 min
   "Lav3_Prog14_EnjIni_NivAg" : Int AT 4x402156, 10 min
   "Lav3_Prog14_EnjIni_Tiempo" : Int AT 4x402157, 10 min
   "Lav3_Prog14_PreLav_NivAg" : Int AT 4x402159, 10 min
   "Lav3_Prog14_PreLav_AgCaliente" : Int AT 4x402160, 10 min
   "Lav3_Prog14_Lav1_NivAg" : Int AT 4x402162, 10 min
   "Lav3_Prog14_Lav1_AgCaliente" : Int AT 4x402163, 10 min
   "Lav3_Prog14_EnjFin_Cant" : Int AT 4x402165, 10 min
   "Lav3_Prog14_Lav2_Tiempo" : Int AT 4x402164, 10 min
   "Lav3_Prog14_Lav2_NivAg" : Int AT 4x402166, 10 min
   "Lav3_Prog14_EnjFin_Tiempo" : Int AT 4x402167, 10 min
   "Lav3_Prog14_Lav2_AgCaliente" : Int AT 4x402168, 10 min
   "Lav3_Prog14_Centr_Tiempo" : Int AT 4x402169, 10 min
   "Lav3_Prog14_PreLav_Vapor" : Int AT 4x402170, 10 min
   "Lav3_Prog14_PreLav_Temperatura" : Int AT 4x402171, 10 min
   "Lav3_Prog14_Lav1_Temperatura" : Int AT 4x402172, 10 min
   "Lav3_Prog14_Lav2_Temperatura" : Int AT 4x401384, 10 min
   "Lav3_Prog14_PreLav_Tiempo" : Int AT 4x402158, 10 min
   "Lav3_Prog14_Lav1_Tiempo" : Int AT 4x402161, 10 min
   "Lav3_Prog15_EnjIni_Cant" : Int AT 4x402219, 10 min
   "Lav3_Prog15_EnjIni_NivAg" : Int AT 4x402220, 10 min
   "Lav3_Prog15_EnjIni_Tiempo" : Int AT 4x402221, 10 min
   "Lav3_Prog15_PreLav_NivAg" : Int AT 4x402223, 10 min
   "Lav3_Prog15_PreLav_AgCaliente" : Int AT 4x402224, 10 min
   "Lav3_Prog15_Lav1_NivAg" : Int AT 4x402226, 10 min
   "Lav3_Prog15_Lav1_AgCaliente" : Int AT 4x402227, 10 min
   "Lav3_Prog15_EnjFin_Cant" : Int AT 4x402229, 10 min
   "Lav3_Prog15_Lav2_Tiempo" : Int AT 4x402228, 10 min
   "Lav3_Prog15_Lav2_NivAg" : Int AT 4x402230, 10 min
   "Lav3_Prog15_EnjFin_Tiempo" : Int AT 4x402231, 10 min
   "Lav3_Prog15_Lav2_AgCaliente" : Int AT 4x402232, 10 min
   "Lav3_Prog15_Centr_Tiempo" : Int AT 4x402233, 10 min
   "Lav3_Prog15_PreLav_Vapor" : Int AT 4x402234, 10 min
   "Lav3_Prog15_PreLav_Temperatura" : Int AT 4x402235, 10 min
   "Lav3_Prog15_Lav1_Temperatura" : Int AT 4x402236, 10 min
   "Lav3_Prog15_Lav2_Temperatura" : Int AT 4x401385, 10 min
   "Lav3_Prog15_PreLav_Tiempo" : Int AT 4x402222, 10 min
   "Lav3_Prog15_Lav1_Tiempo" : Int AT 4x402225, 10 min

HMI tags "ProLav2"
   "Lav2_Prog1_EnjIni_Cant" : Int AT 4x402562, 10 min
   "Lav2_Prog1_EnjIni_NivAg" : Int AT 4x402563, 10 min
   "Lav2_Prog1_EnjIni_Tiempo" : Int AT 4x402564, 10 min
   "Lav2_Prog1_PreLav_NivAg" : Int AT 4x402566, 10 min
   "Lav2_Prog1_PreLav_AgCaliente" : Int AT 4x402567, 10 min
   "Lav2_Prog1_Lav1_NivAg" : Int AT 4x402569, 10 min
   "Lav2_Prog1_Lav1_AgCaliente" : Int AT 4x402570, 10 min
   "Lav2_Prog1_EnjFin_Cant" : Int AT 4x402571, 10 min
   "Lav2_Prog1_Lav2_Tiempo" : Int AT 4x402617, 10 min
   "Lav2_Prog1_Lav2_NivAg" : Int AT 4x402572, 10 min
   "Lav2_Prog1_EnjFin_Tiempo" : Int AT 4x402573, 10 min
   "Lav2_Prog1_Lav2_AgCaliente" : Int AT 4x402574, 10 min
   "Lav2_Prog1_Centr_Tiempo" : Int AT 4x402575, 10 min
   "Lav2_Prog1_PreLav_Vapor" : Int AT 4x402576, 10 min
   "Lav2_Prog1_PreLav_Temperatura" : Int AT 4x402589, 10 min
   "Lav2_Prog1_Lav1_Temperatura" : Int AT 4x402591, 10 min
   "Lav2_Prog1_Lav2_Temperatura" : Int AT 4x401057, 10 min
   "Lav2_Prog1_PreLav_Tiempo" : Int AT 4x402565, 10 min
   "Lav2_Prog1_Lav1_Tiempo" : Int AT 4x402568, 10 min
   "Lav2_Prog2_EnjIni_Cant" : Int AT 4x402626, 10 min
   "Lav2_Prog2_EnjIni_NivAg" : Int AT 4x402627, 10 min
   "Lav2_Prog2_EnjIni_Tiempo" : Int AT 4x402628, 10 min
   "Lav2_Prog2_PreLav_NivAg" : Int AT 4x402630, 10 min
   "Lav2_Prog2_PreLav_AgCaliente" : Int AT 4x402631, 10 min
   "Lav2_Prog2_Lav1_NivAg" : Int AT 4x402633, 10 min
   "Lav2_Prog2_Lav1_AgCaliente" : Int AT 4x402634, 10 min
   "Lav2_Prog2_EnjFin_Cant" : Int AT 4x402635, 10 min
   "Lav2_Prog2_Lav2_Tiempo" : Int AT 4x402618, 10 min
   "Lav2_Prog2_Lav2_NivAg" : Int AT 4x402636, 10 min
   "Lav2_Prog2_EnjFin_Tiempo" : Int AT 4x402637, 10 min
   "Lav2_Prog2_Lav2_AgCaliente" : Int AT 4x402638, 10 min
   "Lav2_Prog2_Centr_Tiempo" : Int AT 4x402639, 10 min
   "Lav2_Prog2_PreLav_Vapor" : Int AT 4x402577, 10 min
   "Lav2_Prog2_PreLav_Temperatura" : Int AT 4x402592, 10 min
   "Lav2_Prog2_Lav1_Temperatura" : Int AT 4x402593, 10 min
   "Lav2_Prog2_Lav2_Temperatura" : Int AT 4x401058, 10 min
   "Lav2_Prog2_PreLav_Tiempo" : Int AT 4x402629, 10 min
   "Lav2_Prog2_Lav1_Tiempo" : Int AT 4x402632, 10 min
   "Lav2_Prog3_EnjIni_Cant" : Int AT 4x402690, 10 min
   "Lav2_Prog3_EnjIni_NivAg" : Int AT 4x402691, 10 min
   "Lav2_Prog3_EnjIni_Tiempo" : Int AT 4x402692, 10 min
   "Lav2_Prog3_PreLav_NivAg" : Int AT 4x402694, 10 min
   "Lav2_Prog3_PreLav_AgCaliente" : Int AT 4x402695, 10 min
   "Lav2_Prog3_Lav1_NivAg" : Int AT 4x402697, 10 min
   "Lav2_Prog3_Lav1_AgCaliente" : Int AT 4x402698, 10 min
   "Lav2_Prog3_EnjFin_Cant" : Int AT 4x402699, 10 min
   "Lav2_Prog3_Lav2_Tiempo" : Int AT 4x402619, 10 min
   "Lav2_Prog3_Lav2_NivAg" : Int AT 4x402700, 10 min
   "Lav2_Prog3_EnjFin_Tiempo" : Int AT 4x402701, 10 min
   "Lav2_Prog3_Lav2_AgCaliente" : Int AT 4x402702, 10 min
   "Lav2_Prog3_Centr_Tiempo" : Int AT 4x402703, 10 min
   "Lav2_Prog3_PreLav_Vapor" : Int AT 4x402579, 10 min
   "Lav2_Prog3_PreLav_Temperatura" : Int AT 4x402595, 10 min
   "Lav2_Prog3_Lav1_Temperatura" : Int AT 4x402597, 10 min
   "Lav2_Prog3_Lav2_Temperatura" : Int AT 4x401059, 10 min
   "Lav2_Prog3_PreLav_Tiempo" : Int AT 4x402693, 10 min
   "Lav2_Prog3_Lav1_Tiempo" : Int AT 4x402696, 10 min
   "Lav2_Prog4_EnjIni_Cant" : Int AT 4x402754, 10 min
   "Lav2_Prog4_EnjIni_NivAg" : Int AT 4x402755, 10 min
   "Lav2_Prog4_EnjIni_Tiempo" : Int AT 4x402756, 10 min
   "Lav2_Prog4_PreLav_NivAg" : Int AT 4x402758, 10 min
   "Lav2_Prog4_PreLav_AgCaliente" : Int AT 4x402759, 10 min
   "Lav2_Prog4_Lav1_NivAg" : Int AT 4x402761, 10 min
   "Lav2_Prog4_Lav1_AgCaliente" : Int AT 4x402762, 10 min
   "Lav2_Prog4_EnjFin_Cant" : Int AT 4x402763, 10 min
   "Lav2_Prog4_Lav2_Tiempo" : Int AT 4x402620, 10 min
   "Lav2_Prog4_Lav2_NivAg" : Int AT 4x402764, 10 min
   "Lav2_Prog4_EnjFin_Tiempo" : Int AT 4x402765, 10 min
   "Lav2_Prog4_Lav2_AgCaliente" : Int AT 4x402766, 10 min
   "Lav2_Prog4_Centr_Tiempo" : Int AT 4x402767, 10 min
   "Lav2_Prog4_PreLav_Vapor" : Int AT 4x402581, 10 min
   "Lav2_Prog4_PreLav_Temperatura" : Int AT 4x402599, 10 min
   "Lav2_Prog4_Lav1_Temperatura" : Int AT 4x402600, 10 min
   "Lav2_Prog4_Lav2_Temperatura" : Int AT 4x401060, 10 min
   "Lav2_Prog4_PreLav_Tiempo" : Int AT 4x402757, 10 min
   "Lav2_Prog4_Lav1_Tiempo" : Int AT 4x402760, 10 min
   "Lav2_Prog5_EnjIni_Cant" : Int AT 4x402818, 10 min
   "Lav2_Prog5_EnjIni_NivAg" : Int AT 4x402819, 10 min
   "Lav2_Prog5_EnjIni_Tiempo" : Int AT 4x402820, 10 min
   "Lav2_Prog5_PreLav_NivAg" : Int AT 4x402822, 10 min
   "Lav2_Prog5_PreLav_AgCaliente" : Int AT 4x402823, 10 min
   "Lav2_Prog5_Lav1_NivAg" : Int AT 4x402825, 10 min
   "Lav2_Prog5_Lav1_AgCaliente" : Int AT 4x402826, 10 min
   "Lav2_Prog5_EnjFin_Cant" : Int AT 4x402827, 10 min
   "Lav2_Prog5_Lav2_Tiempo" : Int AT 4x402621, 10 min
   "Lav2_Prog5_Lav2_NivAg" : Int AT 4x402828, 10 min
   "Lav2_Prog5_EnjFin_Tiempo" : Int AT 4x402829, 10 min
   "Lav2_Prog5_Lav2_AgCaliente" : Int AT 4x402830, 10 min
   "Lav2_Prog5_Centr_Tiempo" : Int AT 4x402831, 10 min
   "Lav2_Prog5_PreLav_Vapor" : Int AT 4x402583, 10 min
   "Lav2_Prog5_PreLav_Temperatura" : Int AT 4x402601, 10 min
   "Lav2_Prog5_Lav1_Temperatura" : Int AT 4x402603, 10 min
   "Lav2_Prog5_Lav2_Temperatura" : Int AT 4x401061, 10 min
   "Lav2_Prog5_PreLav_Tiempo" : Int AT 4x402821, 10 min
   "Lav2_Prog5_Lav1_Tiempo" : Int AT 4x402824, 10 min
   "Lav2_Prog6_EnjIni_Cant" : Int AT 4x402882, 10 min
   "Lav2_Prog6_EnjIni_NivAg" : Int AT 4x402883, 10 min
   "Lav2_Prog6_EnjIni_Tiempo" : Int AT 4x402884, 10 min
   "Lav2_Prog6_PreLav_NivAg" : Int AT 4x402886, 10 min
   "Lav2_Prog6_PreLav_AgCaliente" : Int AT 4x402887, 10 min
   "Lav2_Prog6_Lav1_NivAg" : Int AT 4x402889, 10 min
   "Lav2_Prog6_Lav1_AgCaliente" : Int AT 4x402890, 10 min
   "Lav2_Prog6_EnjFin_Cant" : Int AT 4x402891, 10 min
   "Lav2_Prog6_Lav2_Tiempo" : Int AT 4x402622, 10 min
   "Lav2_Prog6_Lav2_NivAg" : Int AT 4x402892, 10 min
   "Lav2_Prog6_EnjFin_Tiempo" : Int AT 4x402893, 10 min
   "Lav2_Prog6_Lav2_AgCaliente" : Int AT 4x402894, 10 min
   "Lav2_Prog6_Centr_Tiempo" : Int AT 4x402895, 10 min
   "Lav2_Prog6_PreLav_Vapor" : Int AT 4x402585, 10 min
   "Lav2_Prog6_PreLav_Temperatura" : Int AT 4x402605, 10 min
   "Lav2_Prog6_Lav1_Temperatura" : Int AT 4x402607, 10 min
   "Lav2_Prog6_Lav2_Temperatura" : Int AT 4x401062, 10 min
   "Lav2_Prog6_PreLav_Tiempo" : Int AT 4x402885, 10 min
   "Lav2_Prog6_Lav1_Tiempo" : Int AT 4x402888, 10 min
   "Lav2_Prog7_EnjIni_Cant" : Int AT 4x402953, 10 min
   "Lav2_Prog7_EnjIni_NivAg" : Int AT 4x402955, 10 min
   "Lav2_Prog7_EnjIni_Tiempo" : Int AT 4x402956, 10 min
   "Lav2_Prog7_PreLav_NivAg" : Int AT 4x402958, 10 min
   "Lav2_Prog7_PreLav_AgCaliente" : Int AT 4x402959, 10 min
   "Lav2_Prog7_Lav1_NivAg" : Int AT 4x402961, 10 min
   "Lav2_Prog7_Lav1_AgCaliente" : Int AT 4x402962, 10 min
   "Lav2_Prog7_EnjFin_Cant" : Int AT 4x402964, 10 min
   "Lav2_Prog7_Lav2_Tiempo" : Int AT 4x402963, 10 min
   "Lav2_Prog7_Lav2_NivAg" : Int AT 4x402965, 10 min
   "Lav2_Prog7_EnjFin_Tiempo" : Int AT 4x402966, 10 min
   "Lav2_Prog7_Lav2_AgCaliente" : Int AT 4x402967, 10 min
   "Lav2_Prog7_Centr_Tiempo" : Int AT 4x402968, 10 min
   "Lav2_Prog7_PreLav_Vapor" : Int AT 4x402969, 10 min
   "Lav2_Prog7_PreLav_Temperatura" : Int AT 4x402970, 10 min
   "Lav2_Prog7_Lav1_Temperatura" : Int AT 4x402971, 10 min
   "Lav2_Prog7_Lav2_Temperatura" : Int AT 4x401121, 10 min
   "Lav2_Prog7_PreLav_Tiempo" : Int AT 4x402957, 10 min
   "Lav2_Prog7_Lav1_Tiempo" : Int AT 4x402960, 10 min
   "Lav2_Prog8_EnjIni_Cant" : Int AT 4x402978, 10 min
   "Lav2_Prog8_EnjIni_NivAg" : Int AT 4x402979, 10 min
   "Lav2_Prog8_EnjIni_Tiempo" : Int AT 4x402980, 10 min
   "Lav2_Prog8_PreLav_NivAg" : Int AT 4x402982, 10 min
   "Lav2_Prog8_PreLav_AgCaliente" : Int AT 4x402983, 10 min
   "Lav2_Prog8_Lav1_NivAg" : Int AT 4x402985, 10 min
   "Lav2_Prog8_Lav1_AgCaliente" : Int AT 4x402986, 10 min
   "Lav2_Prog8_EnjFin_Cant" : Int AT 4x402988, 10 min
   "Lav2_Prog8_Lav2_Tiempo" : Int AT 4x402987, 10 min
   "Lav2_Prog8_Lav2_NivAg" : Int AT 4x402989, 10 min
   "Lav2_Prog8_EnjFin_Tiempo" : Int AT 4x402990, 10 min
   "Lav2_Prog8_Lav2_AgCaliente" : Int AT 4x402991, 10 min
   "Lav2_Prog8_Centr_Tiempo" : Int AT 4x402992, 10 min
   "Lav2_Prog8_PreLav_Vapor" : Int AT 4x402993, 10 min
   "Lav2_Prog8_PreLav_Temperatura" : Int AT 4x402994, 10 min
   "Lav2_Prog8_Lav1_Temperatura" : Int AT 4x402995, 10 min
   "Lav2_Prog8_Lav2_Temperatura" : Int AT 4x401186, 10 min
   "Lav2_Prog8_PreLav_Tiempo" : Int AT 4x402981, 10 min
   "Lav2_Prog8_Lav1_Tiempo" : Int AT 4x402984, 10 min
   "Lav2_Prog9_EnjIni_Cant" : Int AT 4x402996, 10 min
   "Lav2_Prog9_EnjIni_NivAg" : Int AT 4x402997, 10 min
   "Lav2_Prog9_EnjIni_Tiempo" : Int AT 4x402998, 10 min
   "Lav2_Prog9_PreLav_NivAg" : Int AT 4x403000, 10 min
   "Lav2_Prog9_PreLav_AgCaliente" : Int AT 4x403001, 10 min
   "Lav2_Prog9_Lav1_NivAg" : Int AT 4x403003, 10 min
   "Lav2_Prog9_Lav1_AgCaliente" : Int AT 4x403004, 10 min
   "Lav2_Prog9_EnjFin_Cant" : Int AT 4x403006, 10 min
   "Lav2_Prog9_Lav2_Tiempo" : Int AT 4x403005, 10 min
   "Lav2_Prog9_Lav2_NivAg" : Int AT 4x403007, 10 min
   "Lav2_Prog9_EnjFin_Tiempo" : Int AT 4x403008, 10 min
   "Lav2_Prog9_Lav2_AgCaliente" : Int AT 4x403009, 10 min
   "Lav2_Prog9_Centr_Tiempo" : Int AT 4x403010, 10 min
   "Lav2_Prog9_PreLav_Vapor" : Int AT 4x403011, 10 min
   "Lav2_Prog9_PreLav_Temperatura" : Int AT 4x403012, 10 min
   "Lav2_Prog9_Lav1_Temperatura" : Int AT 4x403013, 10 min
   "Lav2_Prog9_Lav2_Temperatura" : Int AT 4x401251, 10 min
   "Lav2_Prog9_PreLav_Tiempo" : Int AT 4x402999, 10 min
   "Lav2_Prog9_Lav1_Tiempo" : Int AT 4x403002, 10 min
   "Lav2_Prog10_EnjIni_Cant" : Int AT 4x403014, 10 min
   "Lav2_Prog10_EnjIni_NivAg" : Int AT 4x403015, 10 min
   "Lav2_Prog10_EnjIni_Tiempo" : Int AT 4x403016, 10 min
   "Lav2_Prog10_PreLav_NivAg" : Int AT 4x403018, 10 min
   "Lav2_Prog10_PreLav_AgCaliente" : Int AT 4x403019, 10 min
   "Lav2_Prog10_Lav1_NivAg" : Int AT 4x403021, 10 min
   "Lav2_Prog10_Lav1_AgCaliente" : Int AT 4x403022, 10 min
   "Lav2_Prog10_EnjFin_Cant" : Int AT 4x403024, 10 min
   "Lav2_Prog10_Lav2_Tiempo" : Int AT 4x403023, 10 min
   "Lav2_Prog10_Lav2_NivAg" : Int AT 4x403025, 10 min
   "Lav2_Prog10_EnjFin_Tiempo" : Int AT 4x403026, 10 min
   "Lav2_Prog10_Lav2_AgCaliente" : Int AT 4x403027, 10 min
   "Lav2_Prog10_Centr_Tiempo" : Int AT 4x403028, 10 min
   "Lav2_Prog10_PreLav_Vapor" : Int AT 4x403029, 10 min
   "Lav2_Prog10_PreLav_Temperatura" : Int AT 4x403030, 10 min
   "Lav2_Prog10_Lav1_Temperatura" : Int AT 4x403031, 10 min
   "Lav2_Prog10_Lav2_Temperatura" : Int AT 4x401316, 10 min
   "Lav2_Prog10_PreLav_Tiempo" : Int AT 4x403017, 10 min
   "Lav2_Prog10_Lav1_Tiempo" : Int AT 4x403020, 10 min
   "Lav2_Prog11_EnjIni_Cant" : Int AT 4x403033, 10 min
   "Lav2_Prog11_EnjIni_NivAg" : Int AT 4x403034, 10 min
   "Lav2_Prog11_EnjIni_Tiempo" : Int AT 4x403035, 10 min
   "Lav2_Prog11_PreLav_NivAg" : Int AT 4x403037, 10 min
   "Lav2_Prog11_PreLav_AgCaliente" : Int AT 4x403038, 10 min
   "Lav2_Prog11_Lav1_NivAg" : Int AT 4x403040, 10 min
   "Lav2_Prog11_Lav1_AgCaliente" : Int AT 4x403041, 10 min
   "Lav2_Prog11_EnjFin_Cant" : Int AT 4x403043, 10 min
   "Lav2_Prog11_Lav2_Tiempo" : Int AT 4x403042, 10 min
   "Lav2_Prog11_Lav2_NivAg" : Int AT 4x403044, 10 min
   "Lav2_Prog11_EnjFin_Tiempo" : Int AT 4x403045, 10 min
   "Lav2_Prog11_Lav2_AgCaliente" : Int AT 4x403046, 10 min
   "Lav2_Prog11_Centr_Tiempo" : Int AT 4x403047, 10 min
   "Lav2_Prog11_PreLav_Vapor" : Int AT 4x403048, 10 min
   "Lav2_Prog11_PreLav_Temperatura" : Int AT 4x403049, 10 min
   "Lav2_Prog11_Lav1_Temperatura" : Int AT 4x403050, 10 min
   "Lav2_Prog11_Lav2_Temperatura" : Int AT 4x401381, 10 min
   "Lav2_Prog11_PreLav_Tiempo" : Int AT 4x403036, 10 min
   "Lav2_Prog11_Lav1_Tiempo" : Int AT 4x403039, 10 min
   "Lav2_Prog12_EnjIni_Cant" : Int AT 4x403051, 10 min
   "Lav2_Prog12_EnjIni_NivAg" : Int AT 4x403052, 10 min
   "Lav2_Prog12_EnjIni_Tiempo" : Int AT 4x403053, 10 min
   "Lav2_Prog12_PreLav_NivAg" : Int AT 4x403055, 10 min
   "Lav2_Prog12_PreLav_AgCaliente" : Int AT 4x403056, 10 min
   "Lav2_Prog12_Lav1_NivAg" : Int AT 4x403058, 10 min
   "Lav2_Prog12_Lav1_AgCaliente" : Int AT 4x403059, 10 min
   "Lav2_Prog12_EnjFin_Cant" : Int AT 4x403061, 10 min
   "Lav2_Prog12_Lav2_Tiempo" : Int AT 4x403060, 10 min
   "Lav2_Prog12_Lav2_NivAg" : Int AT 4x403062, 10 min
   "Lav2_Prog12_EnjFin_Tiempo" : Int AT 4x403063, 10 min
   "Lav2_Prog12_Lav2_AgCaliente" : Int AT 4x403064, 10 min
   "Lav2_Prog12_Centr_Tiempo" : Int AT 4x403065, 10 min
   "Lav2_Prog12_PreLav_Vapor" : Int AT 4x403066, 10 min
   "Lav2_Prog12_PreLav_Temperatura" : Int AT 4x403067, 10 min
   "Lav2_Prog12_Lav1_Temperatura" : Int AT 4x403068, 10 min
   "Lav2_Prog12_Lav2_Temperatura" : Int AT 4x401382, 10 min
   "Lav2_Prog12_PreLav_Tiempo" : Int AT 4x403054, 10 min
   "Lav2_Prog12_Lav1_Tiempo" : Int AT 4x403057, 10 min
   "Lav2_Prog13_EnjIni_Cant" : Int AT 4x402091, 10 min
   "Lav2_Prog13_EnjIni_NivAg" : Int AT 4x402092, 10 min
   "Lav2_Prog13_EnjIni_Tiempo" : Int AT 4x402093, 10 min
   "Lav2_Prog13_PreLav_NivAg" : Int AT 4x402095, 10 min
   "Lav2_Prog13_PreLav_AgCaliente" : Int AT 4x402096, 10 min
   "Lav2_Prog13_Lav1_NivAg" : Int AT 4x402098, 10 min
   "Lav2_Prog13_Lav1_AgCaliente" : Int AT 4x402099, 10 min
   "Lav2_Prog13_EnjFin_Cant" : Int AT 4x402101, 10 min
   "Lav2_Prog13_Lav2_Tiempo" : Int AT 4x402100, 10 min
   "Lav2_Prog13_Lav2_NivAg" : Int AT 4x402102, 10 min
   "Lav2_Prog13_EnjFin_Tiempo" : Int AT 4x402103, 10 min
   "Lav2_Prog13_Lav2_AgCaliente" : Int AT 4x402104, 10 min
   "Lav2_Prog13_Centr_Tiempo" : Int AT 4x402105, 10 min
   "Lav2_Prog13_PreLav_Vapor" : Int AT 4x402106, 10 min
   "Lav2_Prog13_PreLav_Temperatura" : Int AT 4x402107, 10 min
   "Lav2_Prog13_Lav1_Temperatura" : Int AT 4x402108, 10 min
   "Lav2_Prog13_Lav2_Temperatura" : Int AT 4x401383, 10 min
   "Lav2_Prog13_PreLav_Tiempo" : Int AT 4x402094, 10 min
   "Lav2_Prog13_Lav1_Tiempo" : Int AT 4x402097, 10 min
   "Lav2_Prog14_EnjIni_Cant" : Int AT 4x402155, 10 min
   "Lav2_Prog14_EnjIni_NivAg" : Int AT 4x402156, 10 min
   "Lav2_Prog14_EnjIni_Tiempo" : Int AT 4x402157, 10 min
   "Lav2_Prog14_PreLav_NivAg" : Int AT 4x402159, 10 min
   "Lav2_Prog14_PreLav_AgCaliente" : Int AT 4x402160, 10 min
   "Lav2_Prog14_Lav1_NivAg" : Int AT 4x402162, 10 min
   "Lav2_Prog14_Lav1_AgCaliente" : Int AT 4x402163, 10 min
   "Lav2_Prog14_EnjFin_Cant" : Int AT 4x402165, 10 min
   "Lav2_Prog14_Lav2_Tiempo" : Int AT 4x402164, 10 min
   "Lav2_Prog14_Lav2_NivAg" : Int AT 4x402166, 10 min
   "Lav2_Prog14_EnjFin_Tiempo" : Int AT 4x402167, 10 min
   "Lav2_Prog14_Lav2_AgCaliente" : Int AT 4x402168, 10 min
   "Lav2_Prog14_Centr_Tiempo" : Int AT 4x402169, 10 min
   "Lav2_Prog14_PreLav_Vapor" : Int AT 4x402170, 10 min
   "Lav2_Prog14_PreLav_Temperatura" : Int AT 4x402171, 10 min
   "Lav2_Prog14_Lav1_Temperatura" : Int AT 4x402172, 10 min
   "Lav2_Prog14_Lav2_Temperatura" : Int AT 4x401384, 10 min
   "Lav2_Prog14_PreLav_Tiempo" : Int AT 4x402158, 10 min
   "Lav2_Prog14_Lav1_Tiempo" : Int AT 4x402161, 10 min
   "Lav2_Prog15_EnjIni_Cant" : Int AT 4x402219, 10 min
   "Lav2_Prog15_EnjIni_NivAg" : Int AT 4x402220, 10 min
   "Lav2_Prog15_EnjIni_Tiempo" : Int AT 4x402221, 10 min
   "Lav2_Prog15_PreLav_NivAg" : Int AT 4x402223, 10 min
   "Lav2_Prog15_PreLav_AgCaliente" : Int AT 4x402224, 10 min
   "Lav2_Prog15_Lav1_NivAg" : Int AT 4x402226, 10 min
   "Lav2_Prog15_Lav1_AgCaliente" : Int AT 4x402227, 10 min
   "Lav2_Prog15_EnjFin_Cant" : Int AT 4x402229, 10 min
   "Lav2_Prog15_Lav2_Tiempo" : Int AT 4x402228, 10 min
   "Lav2_Prog15_Lav2_NivAg" : Int AT 4x402230, 10 min
   "Lav2_Prog15_EnjFin_Tiempo" : Int AT 4x402231, 10 min
   "Lav2_Prog15_Lav2_AgCaliente" : Int AT 4x402232, 10 min
   "Lav2_Prog15_Centr_Tiempo" : Int AT 4x402233, 10 min
   "Lav2_Prog15_PreLav_Vapor" : Int AT 4x402234, 10 min
   "Lav2_Prog15_PreLav_Temperatura" : Int AT 4x402235, 10 min
   "Lav2_Prog15_Lav1_Temperatura" : Int AT 4x402236, 10 min
   "Lav2_Prog15_Lav2_Temperatura" : Int AT 4x401385, 10 min
   "Lav2_Prog15_PreLav_Tiempo" : Int AT 4x402222, 10 min
   "Lav2_Prog15_Lav1_Tiempo" : Int AT 4x402225, 10 min

